REGION Network 19: Panel 19
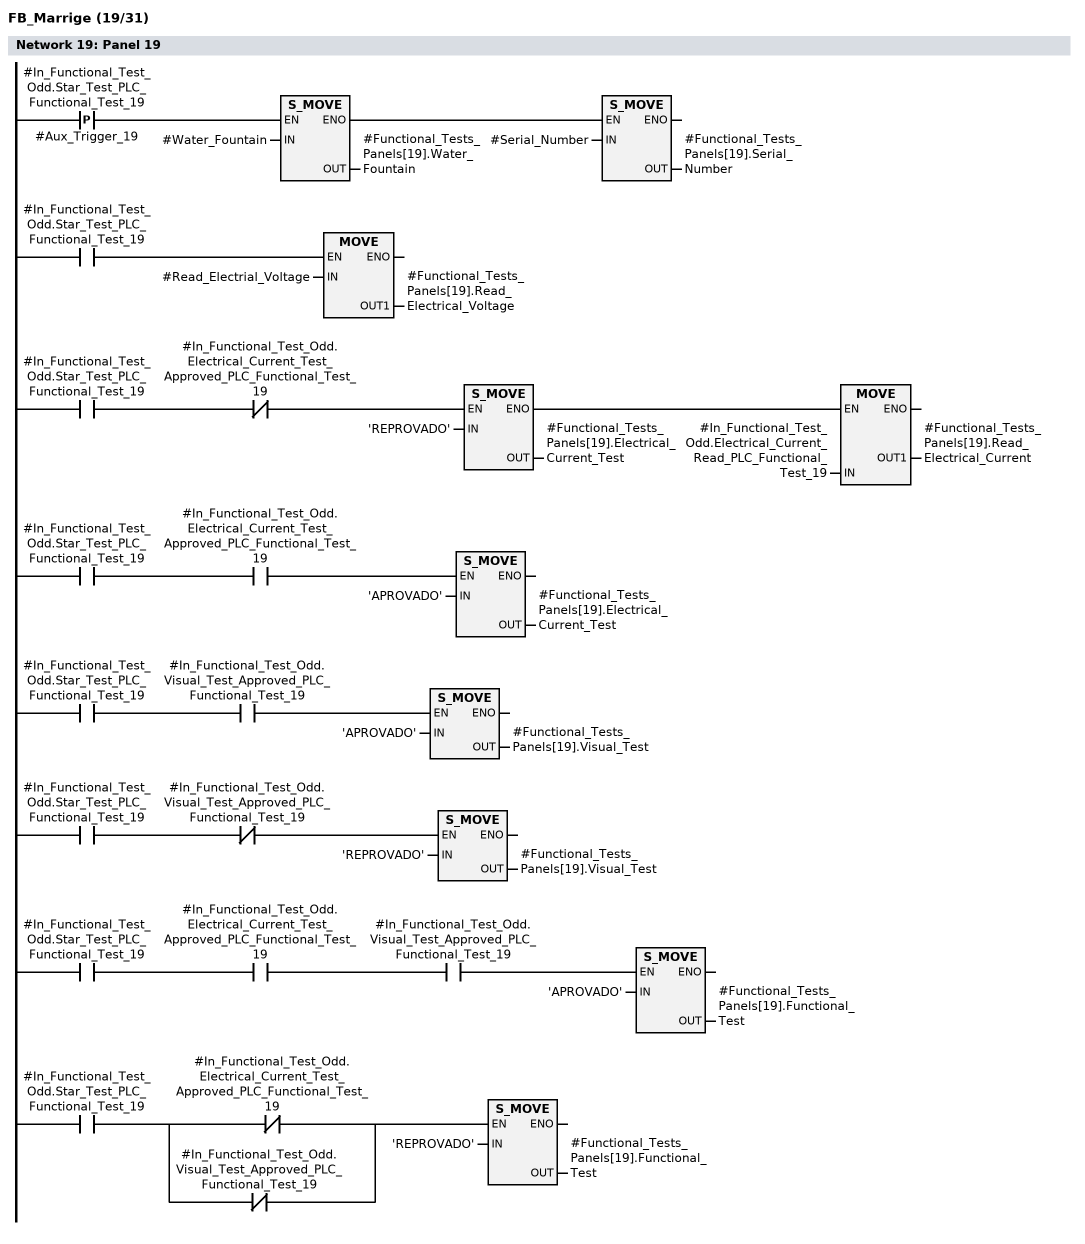
   RUNG wire#powerrail
      P_Contact(operand := #In_Functional_Test_Odd.Star_Test_PLC_Functional_Test_19, bit := #Aux_Trigger_19)
      S_Move(in := #Water_Fountain, out => #Functional_Tests_Panels[19].Water_Fountain)
      S_Move(in := #Serial_Number, out => #Functional_Tests_Panels[19].Serial_Number)
   END_RUNG
   RUNG wire#powerrail
      Contact( #In_Functional_Test_Odd.Star_Test_PLC_Functional_Test_19 )
      Move(in := #Read_Electrial_Voltage, out1 => #Functional_Tests_Panels[19].Read_Electrical_Voltage)
   END_RUNG
   RUNG wire#powerrail
      Contact( #In_Functional_Test_Odd.Star_Test_PLC_Functional_Test_19 )
      I_Contact( #In_Functional_Test_Odd.Electrical_Current_Test_Approved_PLC_Functional_Test_19 )
      S_Move(in := 'REPROVADO', out => #Functional_Tests_Panels[19].Electrical_Current_Test)
      Move(in := #In_Functional_Test_Odd.Electrical_Current_Read_PLC_Functional_Test_19, out1 => #Functional_Tests_Panels[19].Read_Electrical_Current)
   END_RUNG
   RUNG wire#powerrail
      Contact( #In_Functional_Test_Odd.Star_Test_PLC_Functional_Test_19 )
      Contact( #In_Functional_Test_Odd.Electrical_Current_Test_Approved_PLC_Functional_Test_19 )
      S_Move(in := 'APROVADO', out => #Functional_Tests_Panels[19].Electrical_Current_Test)
   END_RUNG
   RUNG wire#powerrail
      Contact( #In_Functional_Test_Odd.Star_Test_PLC_Functional_Test_19 )
      Contact( #In_Functional_Test_Odd.Visual_Test_Approved_PLC_Functional_Test_19 )
      S_Move(in := 'APROVADO', out => #Functional_Tests_Panels[19].Visual_Test)
   END_RUNG
   RUNG wire#powerrail
      Contact( #In_Functional_Test_Odd.Star_Test_PLC_Functional_Test_19 )
      I_Contact( #In_Functional_Test_Odd.Visual_Test_Approved_PLC_Functional_Test_19 )
      S_Move(in := 'REPROVADO', out => #Functional_Tests_Panels[19].Visual_Test)
   END_RUNG
   RUNG wire#powerrail
      Contact( #In_Functional_Test_Odd.Star_Test_PLC_Functional_Test_19 )
      Contact( #In_Functional_Test_Odd.Electrical_Current_Test_Approved_PLC_Functional_Test_19 )
      Contact( #In_Functional_Test_Odd.Visual_Test_Approved_PLC_Functional_Test_19 )
      S_Move(in := 'APROVADO', out => #Functional_Tests_Panels[19].Functional_Test)
   END_RUNG
   RUNG wire#powerrail
      Contact( #In_Functional_Test_Odd.Star_Test_PLC_Functional_Test_19 )
      wire#w1
      I_Contact( #In_Functional_Test_Odd.Electrical_Current_Test_Approved_PLC_Functional_Test_19 )
      wire#w2
      S_Move(in := 'REPROVADO', out => #Functional_Tests_Panels[19].Functional_Test)
   END_RUNG
   RUNG wire#w1
      I_Contact( #In_Functional_Test_Odd.Visual_Test_Approved_PLC_Functional_Test_19 )
   END_RUNG wire#w2
   // the same network as SCL:
   #_w1 := #In_Functional_Test_Odd.Star_Test_PLC_Functional_Test_19 AND NOT #Aux_Trigger_19;   // rising edge of #In_Functional_Test_Odd.Star_Test_PLC_Functional_Test_19
   #Aux_Trigger_19 := #In_Functional_Test_Odd.Star_Test_PLC_Functional_Test_19;
   IF #_w1 THEN
       #Functional_Tests_Panels[19].Water_Fountain := #Water_Fountain;
       #Functional_Tests_Panels[19].Serial_Number := #Serial_Number;
   END_IF;
   IF #In_Functional_Test_Odd.Star_Test_PLC_Functional_Test_19 THEN
       #Functional_Tests_Panels[19].Read_Electrical_Voltage := #Read_Electrial_Voltage;
   END_IF;
   IF #In_Functional_Test_Odd.Star_Test_PLC_Functional_Test_19 AND NOT #In_Functional_Test_Odd.Electrical_Current_Test_Approved_PLC_Functional_Test_19 THEN
       #Functional_Tests_Panels[19].Electrical_Current_Test := 'REPROVADO';
       #Functional_Tests_Panels[19].Read_Electrical_Current := #In_Functional_Test_Odd.Electrical_Current_Read_PLC_Functional_Test_19;
   END_IF;
   IF #In_Functional_Test_Odd.Star_Test_PLC_Functional_Test_19 AND #In_Functional_Test_Odd.Electrical_Current_Test_Approved_PLC_Functional_Test_19 THEN
       #Functional_Tests_Panels[19].Electrical_Current_Test := 'APROVADO';
   END_IF;
   IF #In_Functional_Test_Odd.Star_Test_PLC_Functional_Test_19 AND #In_Functional_Test_Odd.Visual_Test_Approved_PLC_Functional_Test_19 THEN
       #Functional_Tests_Panels[19].Visual_Test := 'APROVADO';
   END_IF;
   IF #In_Functional_Test_Odd.Star_Test_PLC_Functional_Test_19 AND NOT #In_Functional_Test_Odd.Visual_Test_Approved_PLC_Functional_Test_19 THEN
       #Functional_Tests_Panels[19].Visual_Test := 'REPROVADO';
   END_IF;
   IF #In_Functional_Test_Odd.Star_Test_PLC_Functional_Test_19 AND #In_Functional_Test_Odd.Electrical_Current_Test_Approved_PLC_Functional_Test_19 AND #In_Functional_Test_Odd.Visual_Test_Approved_PLC_Functional_Test_19 THEN
       #Functional_Tests_Panels[19].Functional_Test := 'APROVADO';
   END_IF;
   IF #In_Functional_Test_Odd.Star_Test_PLC_Functional_Test_19 AND (NOT #In_Functional_Test_Odd.Electrical_Current_Test_Approved_PLC_Functional_Test_19 OR NOT #In_Functional_Test_Odd.Visual_Test_Approved_PLC_Functional_Test_19) THEN
       #Functional_Tests_Panels[19].Functional_Test := 'REPROVADO';
   END_IF;
END_REGION

REGION Network 20: Panel 20
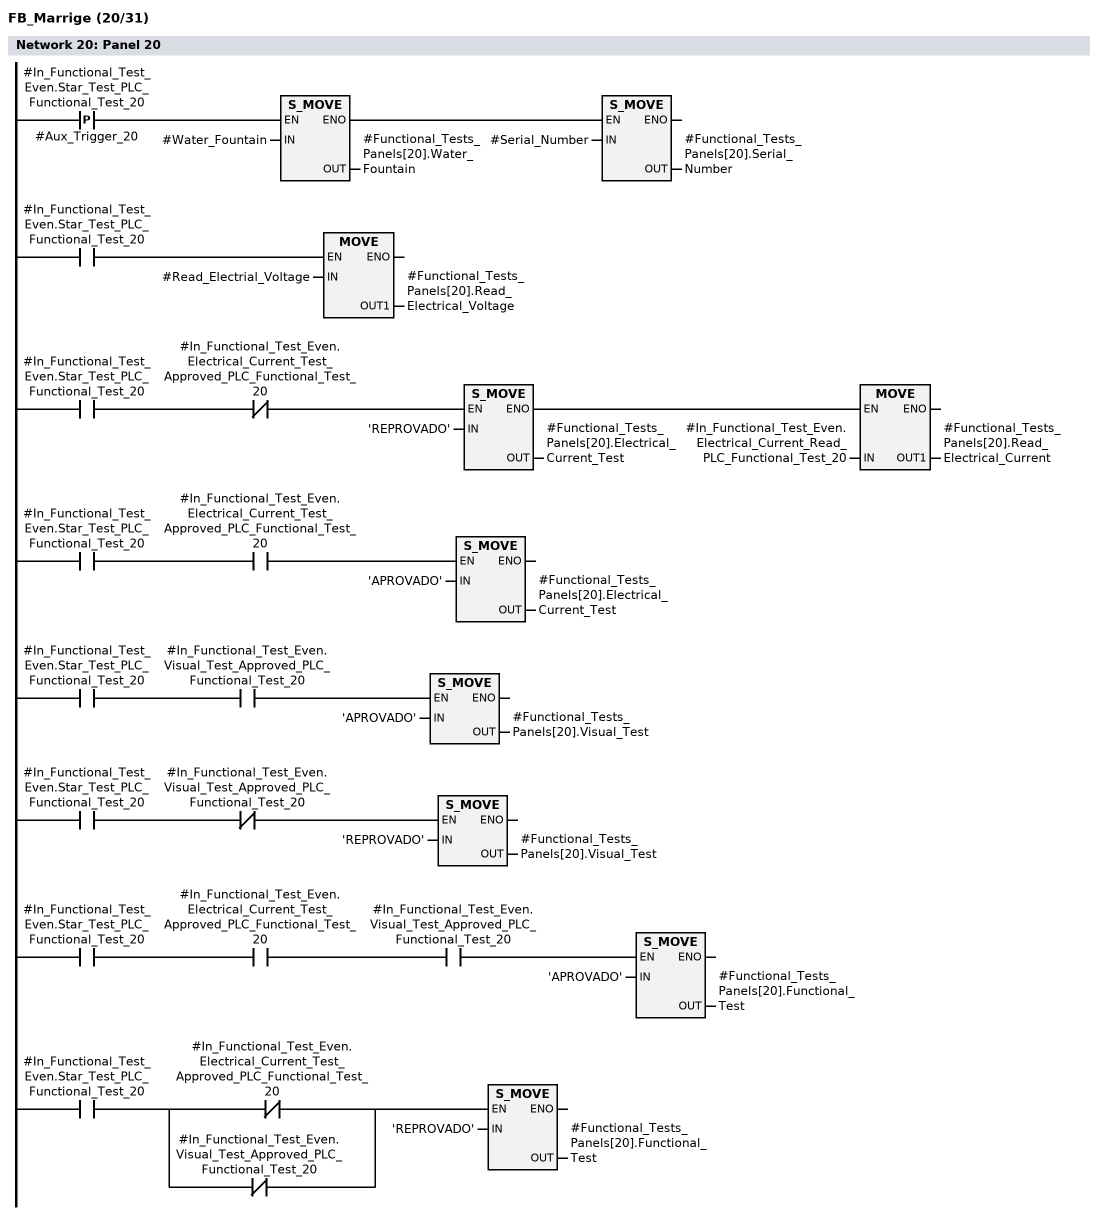
   RUNG wire#powerrail
      P_Contact(operand := #In_Functional_Test_Even.Star_Test_PLC_Functional_Test_20, bit := #Aux_Trigger_20)
      S_Move(in := #Water_Fountain, out => #Functional_Tests_Panels[20].Water_Fountain)
      S_Move(in := #Serial_Number, out => #Functional_Tests_Panels[20].Serial_Number)
   END_RUNG
   RUNG wire#powerrail
      Contact( #In_Functional_Test_Even.Star_Test_PLC_Functional_Test_20 )
      Move(in := #Read_Electrial_Voltage, out1 => #Functional_Tests_Panels[20].Read_Electrical_Voltage)
   END_RUNG
   RUNG wire#powerrail
      Contact( #In_Functional_Test_Even.Star_Test_PLC_Functional_Test_20 )
      I_Contact( #In_Functional_Test_Even.Electrical_Current_Test_Approved_PLC_Functional_Test_20 )
      S_Move(in := 'REPROVADO', out => #Functional_Tests_Panels[20].Electrical_Current_Test)
      Move(in := #In_Functional_Test_Even.Electrical_Current_Read_PLC_Functional_Test_20, out1 => #Functional_Tests_Panels[20].Read_Electrical_Current)
   END_RUNG
   RUNG wire#powerrail
      Contact( #In_Functional_Test_Even.Star_Test_PLC_Functional_Test_20 )
      Contact( #In_Functional_Test_Even.Electrical_Current_Test_Approved_PLC_Functional_Test_20 )
      S_Move(in := 'APROVADO', out => #Functional_Tests_Panels[20].Electrical_Current_Test)
   END_RUNG
   RUNG wire#powerrail
      Contact( #In_Functional_Test_Even.Star_Test_PLC_Functional_Test_20 )
      Contact( #In_Functional_Test_Even.Visual_Test_Approved_PLC_Functional_Test_20 )
      S_Move(in := 'APROVADO', out => #Functional_Tests_Panels[20].Visual_Test)
   END_RUNG
   RUNG wire#powerrail
      Contact( #In_Functional_Test_Even.Star_Test_PLC_Functional_Test_20 )
      I_Contact( #In_Functional_Test_Even.Visual_Test_Approved_PLC_Functional_Test_20 )
      S_Move(in := 'REPROVADO', out => #Functional_Tests_Panels[20].Visual_Test)
   END_RUNG
   RUNG wire#powerrail
      Contact( #In_Functional_Test_Even.Star_Test_PLC_Functional_Test_20 )
      Contact( #In_Functional_Test_Even.Electrical_Current_Test_Approved_PLC_Functional_Test_20 )
      Contact( #In_Functional_Test_Even.Visual_Test_Approved_PLC_Functional_Test_20 )
      S_Move(in := 'APROVADO', out => #Functional_Tests_Panels[20].Functional_Test)
   END_RUNG
   RUNG wire#powerrail
      Contact( #In_Functional_Test_Even.Star_Test_PLC_Functional_Test_20 )
      wire#w1
      I_Contact( #In_Functional_Test_Even.Electrical_Current_Test_Approved_PLC_Functional_Test_20 )
      wire#w2
      S_Move(in := 'REPROVADO', out => #Functional_Tests_Panels[20].Functional_Test)
   END_RUNG
   RUNG wire#w1
      I_Contact( #In_Functional_Test_Even.Visual_Test_Approved_PLC_Functional_Test_20 )
   END_RUNG wire#w2
   // the same network as SCL:
   #_w1 := #In_Functional_Test_Even.Star_Test_PLC_Functional_Test_20 AND NOT #Aux_Trigger_20;   // rising edge of #In_Functional_Test_Even.Star_Test_PLC_Functional_Test_20
   #Aux_Trigger_20 := #In_Functional_Test_Even.Star_Test_PLC_Functional_Test_20;
   IF #_w1 THEN
       #Functional_Tests_Panels[20].Water_Fountain := #Water_Fountain;
       #Functional_Tests_Panels[20].Serial_Number := #Serial_Number;
   END_IF;
   IF #In_Functional_Test_Even.Star_Test_PLC_Functional_Test_20 THEN
       #Functional_Tests_Panels[20].Read_Electrical_Voltage := #Read_Electrial_Voltage;
   END_IF;
   IF #In_Functional_Test_Even.Star_Test_PLC_Functional_Test_20 AND NOT #In_Functional_Test_Even.Electrical_Current_Test_Approved_PLC_Functional_Test_20 THEN
       #Functional_Tests_Panels[20].Electrical_Current_Test := 'REPROVADO';
       #Functional_Tests_Panels[20].Read_Electrical_Current := #In_Functional_Test_Even.Electrical_Current_Read_PLC_Functional_Test_20;
   END_IF;
   IF #In_Functional_Test_Even.Star_Test_PLC_Functional_Test_20 AND #In_Functional_Test_Even.Electrical_Current_Test_Approved_PLC_Functional_Test_20 THEN
       #Functional_Tests_Panels[20].Electrical_Current_Test := 'APROVADO';
   END_IF;
   IF #In_Functional_Test_Even.Star_Test_PLC_Functional_Test_20 AND #In_Functional_Test_Even.Visual_Test_Approved_PLC_Functional_Test_20 THEN
       #Functional_Tests_Panels[20].Visual_Test := 'APROVADO';
   END_IF;
   IF #In_Functional_Test_Even.Star_Test_PLC_Functional_Test_20 AND NOT #In_Functional_Test_Even.Visual_Test_Approved_PLC_Functional_Test_20 THEN
       #Functional_Tests_Panels[20].Visual_Test := 'REPROVADO';
   END_IF;
   IF #In_Functional_Test_Even.Star_Test_PLC_Functional_Test_20 AND #In_Functional_Test_Even.Electrical_Current_Test_Approved_PLC_Functional_Test_20 AND #In_Functional_Test_Even.Visual_Test_Approved_PLC_Functional_Test_20 THEN
       #Functional_Tests_Panels[20].Functional_Test := 'APROVADO';
   END_IF;
   IF #In_Functional_Test_Even.Star_Test_PLC_Functional_Test_20 AND (NOT #In_Functional_Test_Even.Electrical_Current_Test_Approved_PLC_Functional_Test_20 OR NOT #In_Functional_Test_Even.Visual_Test_Approved_PLC_Functional_Test_20) THEN
       #Functional_Tests_Panels[20].Functional_Test := 'REPROVADO';
   END_IF;
END_REGION

REGION Network 21: Panel 21
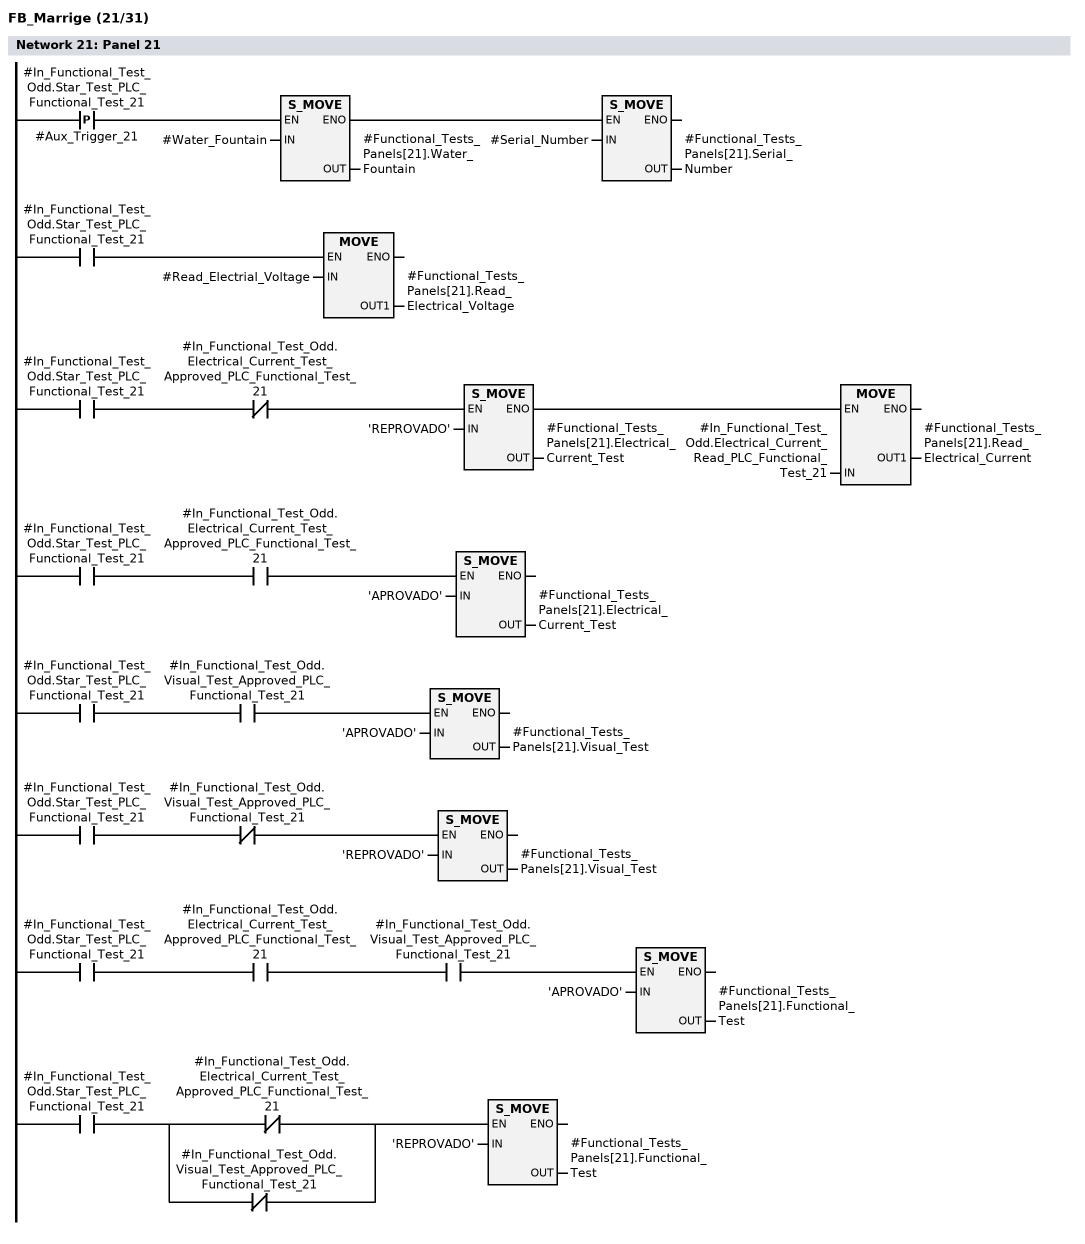
   RUNG wire#powerrail
      P_Contact(operand := #In_Functional_Test_Odd.Star_Test_PLC_Functional_Test_21, bit := #Aux_Trigger_21)
      S_Move(in := #Water_Fountain, out => #Functional_Tests_Panels[21].Water_Fountain)
      S_Move(in := #Serial_Number, out => #Functional_Tests_Panels[21].Serial_Number)
   END_RUNG
   RUNG wire#powerrail
      Contact( #In_Functional_Test_Odd.Star_Test_PLC_Functional_Test_21 )
      Move(in := #Read_Electrial_Voltage, out1 => #Functional_Tests_Panels[21].Read_Electrical_Voltage)
   END_RUNG
   RUNG wire#powerrail
      Contact( #In_Functional_Test_Odd.Star_Test_PLC_Functional_Test_21 )
      I_Contact( #In_Functional_Test_Odd.Electrical_Current_Test_Approved_PLC_Functional_Test_21 )
      S_Move(in := 'REPROVADO', out => #Functional_Tests_Panels[21].Electrical_Current_Test)
      Move(in := #In_Functional_Test_Odd.Electrical_Current_Read_PLC_Functional_Test_21, out1 => #Functional_Tests_Panels[21].Read_Electrical_Current)
   END_RUNG
   RUNG wire#powerrail
      Contact( #In_Functional_Test_Odd.Star_Test_PLC_Functional_Test_21 )
      Contact( #In_Functional_Test_Odd.Electrical_Current_Test_Approved_PLC_Functional_Test_21 )
      S_Move(in := 'APROVADO', out => #Functional_Tests_Panels[21].Electrical_Current_Test)
   END_RUNG
   RUNG wire#powerrail
      Contact( #In_Functional_Test_Odd.Star_Test_PLC_Functional_Test_21 )
      Contact( #In_Functional_Test_Odd.Visual_Test_Approved_PLC_Functional_Test_21 )
      S_Move(in := 'APROVADO', out => #Functional_Tests_Panels[21].Visual_Test)
   END_RUNG
   RUNG wire#powerrail
      Contact( #In_Functional_Test_Odd.Star_Test_PLC_Functional_Test_21 )
      I_Contact( #In_Functional_Test_Odd.Visual_Test_Approved_PLC_Functional_Test_21 )
      S_Move(in := 'REPROVADO', out => #Functional_Tests_Panels[21].Visual_Test)
   END_RUNG
   RUNG wire#powerrail
      Contact( #In_Functional_Test_Odd.Star_Test_PLC_Functional_Test_21 )
      Contact( #In_Functional_Test_Odd.Electrical_Current_Test_Approved_PLC_Functional_Test_21 )
      Contact( #In_Functional_Test_Odd.Visual_Test_Approved_PLC_Functional_Test_21 )
      S_Move(in := 'APROVADO', out => #Functional_Tests_Panels[21].Functional_Test)
   END_RUNG
   RUNG wire#powerrail
      Contact( #In_Functional_Test_Odd.Star_Test_PLC_Functional_Test_21 )
      wire#w1
      I_Contact( #In_Functional_Test_Odd.Electrical_Current_Test_Approved_PLC_Functional_Test_21 )
      wire#w2
      S_Move(in := 'REPROVADO', out => #Functional_Tests_Panels[21].Functional_Test)
   END_RUNG
   RUNG wire#w1
      I_Contact( #In_Functional_Test_Odd.Visual_Test_Approved_PLC_Functional_Test_21 )
   END_RUNG wire#w2
   // the same network as SCL:
   #_w1 := #In_Functional_Test_Odd.Star_Test_PLC_Functional_Test_21 AND NOT #Aux_Trigger_21;   // rising edge of #In_Functional_Test_Odd.Star_Test_PLC_Functional_Test_21
   #Aux_Trigger_21 := #In_Functional_Test_Odd.Star_Test_PLC_Functional_Test_21;
   IF #_w1 THEN
       #Functional_Tests_Panels[21].Water_Fountain := #Water_Fountain;
       #Functional_Tests_Panels[21].Serial_Number := #Serial_Number;
   END_IF;
   IF #In_Functional_Test_Odd.Star_Test_PLC_Functional_Test_21 THEN
       #Functional_Tests_Panels[21].Read_Electrical_Voltage := #Read_Electrial_Voltage;
   END_IF;
   IF #In_Functional_Test_Odd.Star_Test_PLC_Functional_Test_21 AND NOT #In_Functional_Test_Odd.Electrical_Current_Test_Approved_PLC_Functional_Test_21 THEN
       #Functional_Tests_Panels[21].Electrical_Current_Test := 'REPROVADO';
       #Functional_Tests_Panels[21].Read_Electrical_Current := #In_Functional_Test_Odd.Electrical_Current_Read_PLC_Functional_Test_21;
   END_IF;
   IF #In_Functional_Test_Odd.Star_Test_PLC_Functional_Test_21 AND #In_Functional_Test_Odd.Electrical_Current_Test_Approved_PLC_Functional_Test_21 THEN
       #Functional_Tests_Panels[21].Electrical_Current_Test := 'APROVADO';
   END_IF;
   IF #In_Functional_Test_Odd.Star_Test_PLC_Functional_Test_21 AND #In_Functional_Test_Odd.Visual_Test_Approved_PLC_Functional_Test_21 THEN
       #Functional_Tests_Panels[21].Visual_Test := 'APROVADO';
   END_IF;
   IF #In_Functional_Test_Odd.Star_Test_PLC_Functional_Test_21 AND NOT #In_Functional_Test_Odd.Visual_Test_Approved_PLC_Functional_Test_21 THEN
       #Functional_Tests_Panels[21].Visual_Test := 'REPROVADO';
   END_IF;
   IF #In_Functional_Test_Odd.Star_Test_PLC_Functional_Test_21 AND #In_Functional_Test_Odd.Electrical_Current_Test_Approved_PLC_Functional_Test_21 AND #In_Functional_Test_Odd.Visual_Test_Approved_PLC_Functional_Test_21 THEN
       #Functional_Tests_Panels[21].Functional_Test := 'APROVADO';
   END_IF;
   IF #In_Functional_Test_Odd.Star_Test_PLC_Functional_Test_21 AND (NOT #In_Functional_Test_Odd.Electrical_Current_Test_Approved_PLC_Functional_Test_21 OR NOT #In_Functional_Test_Odd.Visual_Test_Approved_PLC_Functional_Test_21) THEN
       #Functional_Tests_Panels[21].Functional_Test := 'REPROVADO';
   END_IF;
END_REGION

REGION Network 22: Panel 22
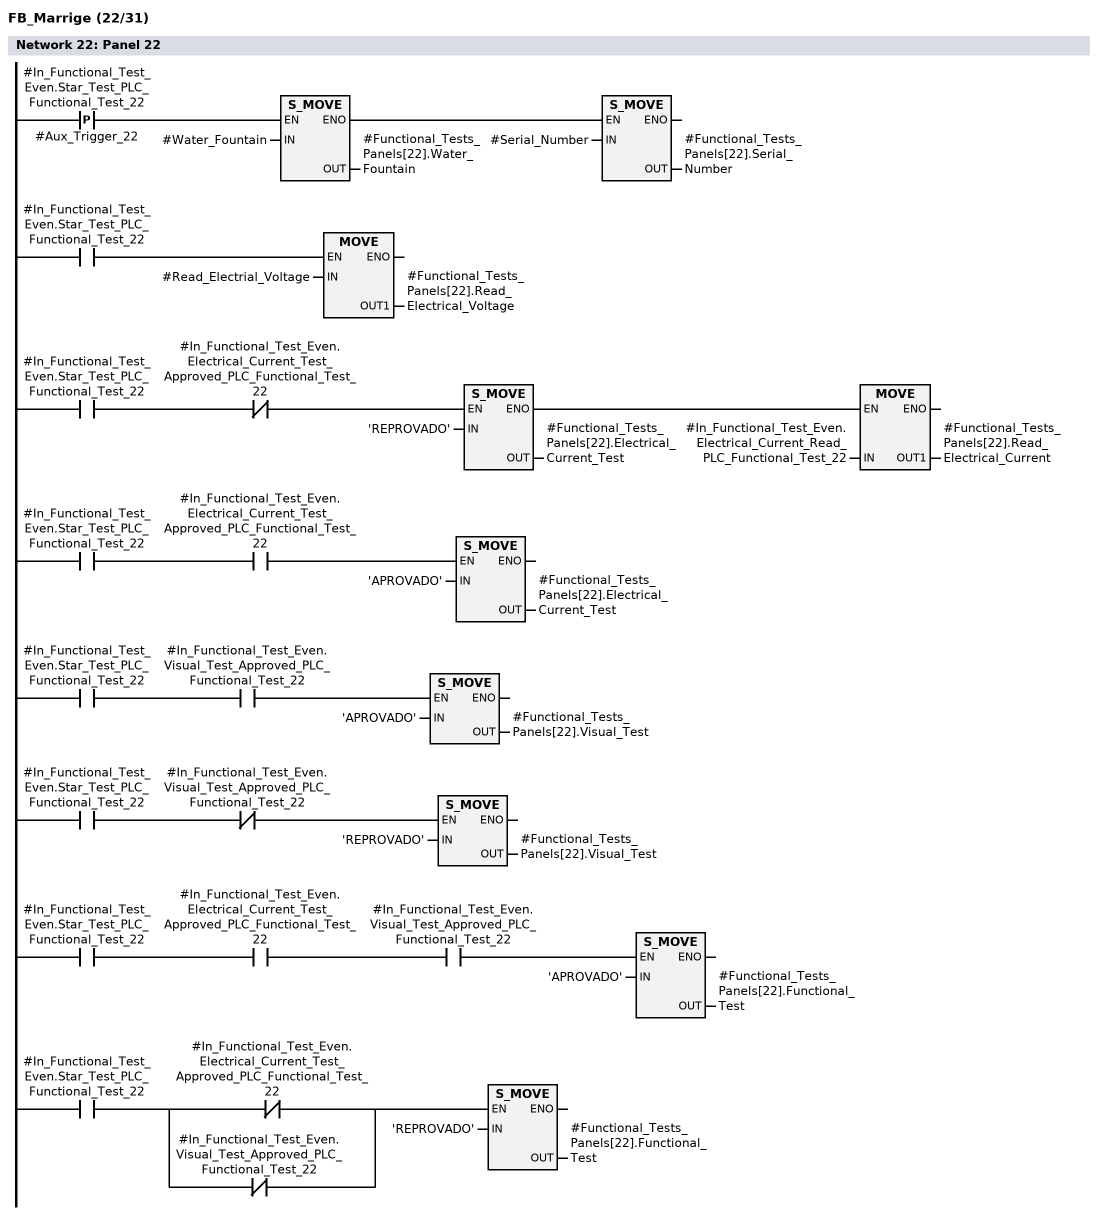
   RUNG wire#powerrail
      P_Contact(operand := #In_Functional_Test_Even.Star_Test_PLC_Functional_Test_22, bit := #Aux_Trigger_22)
      S_Move(in := #Water_Fountain, out => #Functional_Tests_Panels[22].Water_Fountain)
      S_Move(in := #Serial_Number, out => #Functional_Tests_Panels[22].Serial_Number)
   END_RUNG
   RUNG wire#powerrail
      Contact( #In_Functional_Test_Even.Star_Test_PLC_Functional_Test_22 )
      Move(in := #Read_Electrial_Voltage, out1 => #Functional_Tests_Panels[22].Read_Electrical_Voltage)
   END_RUNG
   RUNG wire#powerrail
      Contact( #In_Functional_Test_Even.Star_Test_PLC_Functional_Test_22 )
      I_Contact( #In_Functional_Test_Even.Electrical_Current_Test_Approved_PLC_Functional_Test_22 )
      S_Move(in := 'REPROVADO', out => #Functional_Tests_Panels[22].Electrical_Current_Test)
      Move(in := #In_Functional_Test_Even.Electrical_Current_Read_PLC_Functional_Test_22, out1 => #Functional_Tests_Panels[22].Read_Electrical_Current)
   END_RUNG
   RUNG wire#powerrail
      Contact( #In_Functional_Test_Even.Star_Test_PLC_Functional_Test_22 )
      Contact( #In_Functional_Test_Even.Electrical_Current_Test_Approved_PLC_Functional_Test_22 )
      S_Move(in := 'APROVADO', out => #Functional_Tests_Panels[22].Electrical_Current_Test)
   END_RUNG
   RUNG wire#powerrail
      Contact( #In_Functional_Test_Even.Star_Test_PLC_Functional_Test_22 )
      Contact( #In_Functional_Test_Even.Visual_Test_Approved_PLC_Functional_Test_22 )
      S_Move(in := 'APROVADO', out => #Functional_Tests_Panels[22].Visual_Test)
   END_RUNG
   RUNG wire#powerrail
      Contact( #In_Functional_Test_Even.Star_Test_PLC_Functional_Test_22 )
      I_Contact( #In_Functional_Test_Even.Visual_Test_Approved_PLC_Functional_Test_22 )
      S_Move(in := 'REPROVADO', out => #Functional_Tests_Panels[22].Visual_Test)
   END_RUNG
   RUNG wire#powerrail
      Contact( #In_Functional_Test_Even.Star_Test_PLC_Functional_Test_22 )
      Contact( #In_Functional_Test_Even.Electrical_Current_Test_Approved_PLC_Functional_Test_22 )
      Contact( #In_Functional_Test_Even.Visual_Test_Approved_PLC_Functional_Test_22 )
      S_Move(in := 'APROVADO', out => #Functional_Tests_Panels[22].Functional_Test)
   END_RUNG
   RUNG wire#powerrail
      Contact( #In_Functional_Test_Even.Star_Test_PLC_Functional_Test_22 )
      wire#w1
      I_Contact( #In_Functional_Test_Even.Electrical_Current_Test_Approved_PLC_Functional_Test_22 )
      wire#w2
      S_Move(in := 'REPROVADO', out => #Functional_Tests_Panels[22].Functional_Test)
   END_RUNG
   RUNG wire#w1
      I_Contact( #In_Functional_Test_Even.Visual_Test_Approved_PLC_Functional_Test_22 )
   END_RUNG wire#w2
   // the same network as SCL:
   #_w1 := #In_Functional_Test_Even.Star_Test_PLC_Functional_Test_22 AND NOT #Aux_Trigger_22;   // rising edge of #In_Functional_Test_Even.Star_Test_PLC_Functional_Test_22
   #Aux_Trigger_22 := #In_Functional_Test_Even.Star_Test_PLC_Functional_Test_22;
   IF #_w1 THEN
       #Functional_Tests_Panels[22].Water_Fountain := #Water_Fountain;
       #Functional_Tests_Panels[22].Serial_Number := #Serial_Number;
   END_IF;
   IF #In_Functional_Test_Even.Star_Test_PLC_Functional_Test_22 THEN
       #Functional_Tests_Panels[22].Read_Electrical_Voltage := #Read_Electrial_Voltage;
   END_IF;
   IF #In_Functional_Test_Even.Star_Test_PLC_Functional_Test_22 AND NOT #In_Functional_Test_Even.Electrical_Current_Test_Approved_PLC_Functional_Test_22 THEN
       #Functional_Tests_Panels[22].Electrical_Current_Test := 'REPROVADO';
       #Functional_Tests_Panels[22].Read_Electrical_Current := #In_Functional_Test_Even.Electrical_Current_Read_PLC_Functional_Test_22;
   END_IF;
   IF #In_Functional_Test_Even.Star_Test_PLC_Functional_Test_22 AND #In_Functional_Test_Even.Electrical_Current_Test_Approved_PLC_Functional_Test_22 THEN
       #Functional_Tests_Panels[22].Electrical_Current_Test := 'APROVADO';
   END_IF;
   IF #In_Functional_Test_Even.Star_Test_PLC_Functional_Test_22 AND #In_Functional_Test_Even.Visual_Test_Approved_PLC_Functional_Test_22 THEN
       #Functional_Tests_Panels[22].Visual_Test := 'APROVADO';
   END_IF;
   IF #In_Functional_Test_Even.Star_Test_PLC_Functional_Test_22 AND NOT #In_Functional_Test_Even.Visual_Test_Approved_PLC_Functional_Test_22 THEN
       #Functional_Tests_Panels[22].Visual_Test := 'REPROVADO';
   END_IF;
   IF #In_Functional_Test_Even.Star_Test_PLC_Functional_Test_22 AND #In_Functional_Test_Even.Electrical_Current_Test_Approved_PLC_Functional_Test_22 AND #In_Functional_Test_Even.Visual_Test_Approved_PLC_Functional_Test_22 THEN
       #Functional_Tests_Panels[22].Functional_Test := 'APROVADO';
   END_IF;
   IF #In_Functional_Test_Even.Star_Test_PLC_Functional_Test_22 AND (NOT #In_Functional_Test_Even.Electrical_Current_Test_Approved_PLC_Functional_Test_22 OR NOT #In_Functional_Test_Even.Visual_Test_Approved_PLC_Functional_Test_22) THEN
       #Functional_Tests_Panels[22].Functional_Test := 'REPROVADO';
   END_IF;
END_REGION

REGION Network 23: Panel 23
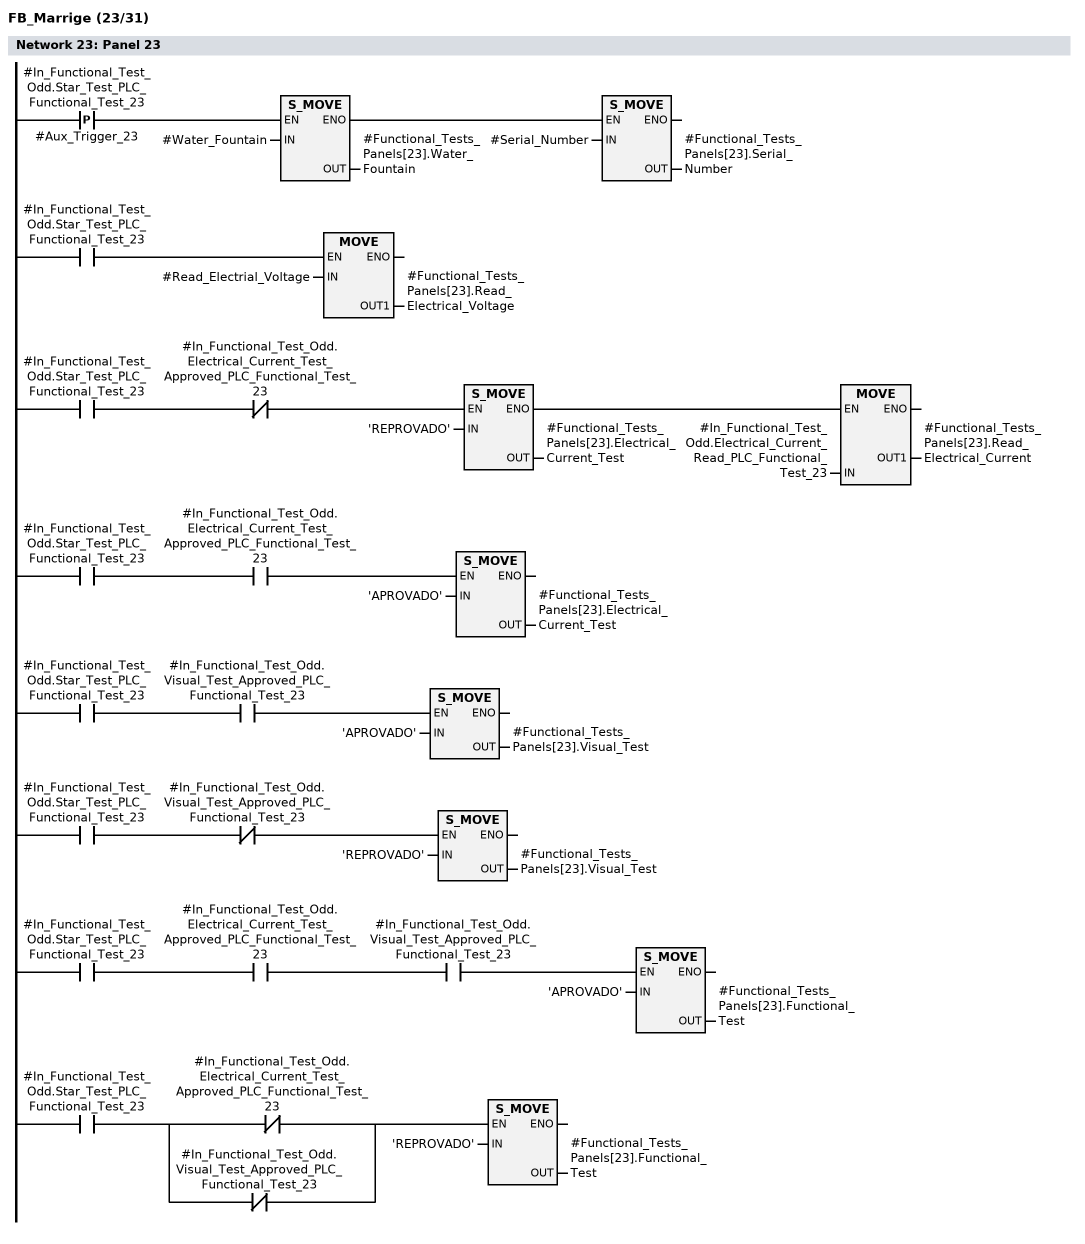
   RUNG wire#powerrail
      P_Contact(operand := #In_Functional_Test_Odd.Star_Test_PLC_Functional_Test_23, bit := #Aux_Trigger_23)
      S_Move(in := #Water_Fountain, out => #Functional_Tests_Panels[23].Water_Fountain)
      S_Move(in := #Serial_Number, out => #Functional_Tests_Panels[23].Serial_Number)
   END_RUNG
   RUNG wire#powerrail
      Contact( #In_Functional_Test_Odd.Star_Test_PLC_Functional_Test_23 )
      Move(in := #Read_Electrial_Voltage, out1 => #Functional_Tests_Panels[23].Read_Electrical_Voltage)
   END_RUNG
   RUNG wire#powerrail
      Contact( #In_Functional_Test_Odd.Star_Test_PLC_Functional_Test_23 )
      I_Contact( #In_Functional_Test_Odd.Electrical_Current_Test_Approved_PLC_Functional_Test_23 )
      S_Move(in := 'REPROVADO', out => #Functional_Tests_Panels[23].Electrical_Current_Test)
      Move(in := #In_Functional_Test_Odd.Electrical_Current_Read_PLC_Functional_Test_23, out1 => #Functional_Tests_Panels[23].Read_Electrical_Current)
   END_RUNG
   RUNG wire#powerrail
      Contact( #In_Functional_Test_Odd.Star_Test_PLC_Functional_Test_23 )
      Contact( #In_Functional_Test_Odd.Electrical_Current_Test_Approved_PLC_Functional_Test_23 )
      S_Move(in := 'APROVADO', out => #Functional_Tests_Panels[23].Electrical_Current_Test)
   END_RUNG
   RUNG wire#powerrail
      Contact( #In_Functional_Test_Odd.Star_Test_PLC_Functional_Test_23 )
      Contact( #In_Functional_Test_Odd.Visual_Test_Approved_PLC_Functional_Test_23 )
      S_Move(in := 'APROVADO', out => #Functional_Tests_Panels[23].Visual_Test)
   END_RUNG
   RUNG wire#powerrail
      Contact( #In_Functional_Test_Odd.Star_Test_PLC_Functional_Test_23 )
      I_Contact( #In_Functional_Test_Odd.Visual_Test_Approved_PLC_Functional_Test_23 )
      S_Move(in := 'REPROVADO', out => #Functional_Tests_Panels[23].Visual_Test)
   END_RUNG
   RUNG wire#powerrail
      Contact( #In_Functional_Test_Odd.Star_Test_PLC_Functional_Test_23 )
      Contact( #In_Functional_Test_Odd.Electrical_Current_Test_Approved_PLC_Functional_Test_23 )
      Contact( #In_Functional_Test_Odd.Visual_Test_Approved_PLC_Functional_Test_23 )
      S_Move(in := 'APROVADO', out => #Functional_Tests_Panels[23].Functional_Test)
   END_RUNG
   RUNG wire#powerrail
      Contact( #In_Functional_Test_Odd.Star_Test_PLC_Functional_Test_23 )
      wire#w1
      I_Contact( #In_Functional_Test_Odd.Electrical_Current_Test_Approved_PLC_Functional_Test_23 )
      wire#w2
      S_Move(in := 'REPROVADO', out => #Functional_Tests_Panels[23].Functional_Test)
   END_RUNG
   RUNG wire#w1
      I_Contact( #In_Functional_Test_Odd.Visual_Test_Approved_PLC_Functional_Test_23 )
   END_RUNG wire#w2
   // the same network as SCL:
   #_w1 := #In_Functional_Test_Odd.Star_Test_PLC_Functional_Test_23 AND NOT #Aux_Trigger_23;   // rising edge of #In_Functional_Test_Odd.Star_Test_PLC_Functional_Test_23
   #Aux_Trigger_23 := #In_Functional_Test_Odd.Star_Test_PLC_Functional_Test_23;
   IF #_w1 THEN
       #Functional_Tests_Panels[23].Water_Fountain := #Water_Fountain;
       #Functional_Tests_Panels[23].Serial_Number := #Serial_Number;
   END_IF;
   IF #In_Functional_Test_Odd.Star_Test_PLC_Functional_Test_23 THEN
       #Functional_Tests_Panels[23].Read_Electrical_Voltage := #Read_Electrial_Voltage;
   END_IF;
   IF #In_Functional_Test_Odd.Star_Test_PLC_Functional_Test_23 AND NOT #In_Functional_Test_Odd.Electrical_Current_Test_Approved_PLC_Functional_Test_23 THEN
       #Functional_Tests_Panels[23].Electrical_Current_Test := 'REPROVADO';
       #Functional_Tests_Panels[23].Read_Electrical_Current := #In_Functional_Test_Odd.Electrical_Current_Read_PLC_Functional_Test_23;
   END_IF;
   IF #In_Functional_Test_Odd.Star_Test_PLC_Functional_Test_23 AND #In_Functional_Test_Odd.Electrical_Current_Test_Approved_PLC_Functional_Test_23 THEN
       #Functional_Tests_Panels[23].Electrical_Current_Test := 'APROVADO';
   END_IF;
   IF #In_Functional_Test_Odd.Star_Test_PLC_Functional_Test_23 AND #In_Functional_Test_Odd.Visual_Test_Approved_PLC_Functional_Test_23 THEN
       #Functional_Tests_Panels[23].Visual_Test := 'APROVADO';
   END_IF;
   IF #In_Functional_Test_Odd.Star_Test_PLC_Functional_Test_23 AND NOT #In_Functional_Test_Odd.Visual_Test_Approved_PLC_Functional_Test_23 THEN
       #Functional_Tests_Panels[23].Visual_Test := 'REPROVADO';
   END_IF;
   IF #In_Functional_Test_Odd.Star_Test_PLC_Functional_Test_23 AND #In_Functional_Test_Odd.Electrical_Current_Test_Approved_PLC_Functional_Test_23 AND #In_Functional_Test_Odd.Visual_Test_Approved_PLC_Functional_Test_23 THEN
       #Functional_Tests_Panels[23].Functional_Test := 'APROVADO';
   END_IF;
   IF #In_Functional_Test_Odd.Star_Test_PLC_Functional_Test_23 AND (NOT #In_Functional_Test_Odd.Electrical_Current_Test_Approved_PLC_Functional_Test_23 OR NOT #In_Functional_Test_Odd.Visual_Test_Approved_PLC_Functional_Test_23) THEN
       #Functional_Tests_Panels[23].Functional_Test := 'REPROVADO';
   END_IF;
END_REGION

REGION Network 24: Panel 24
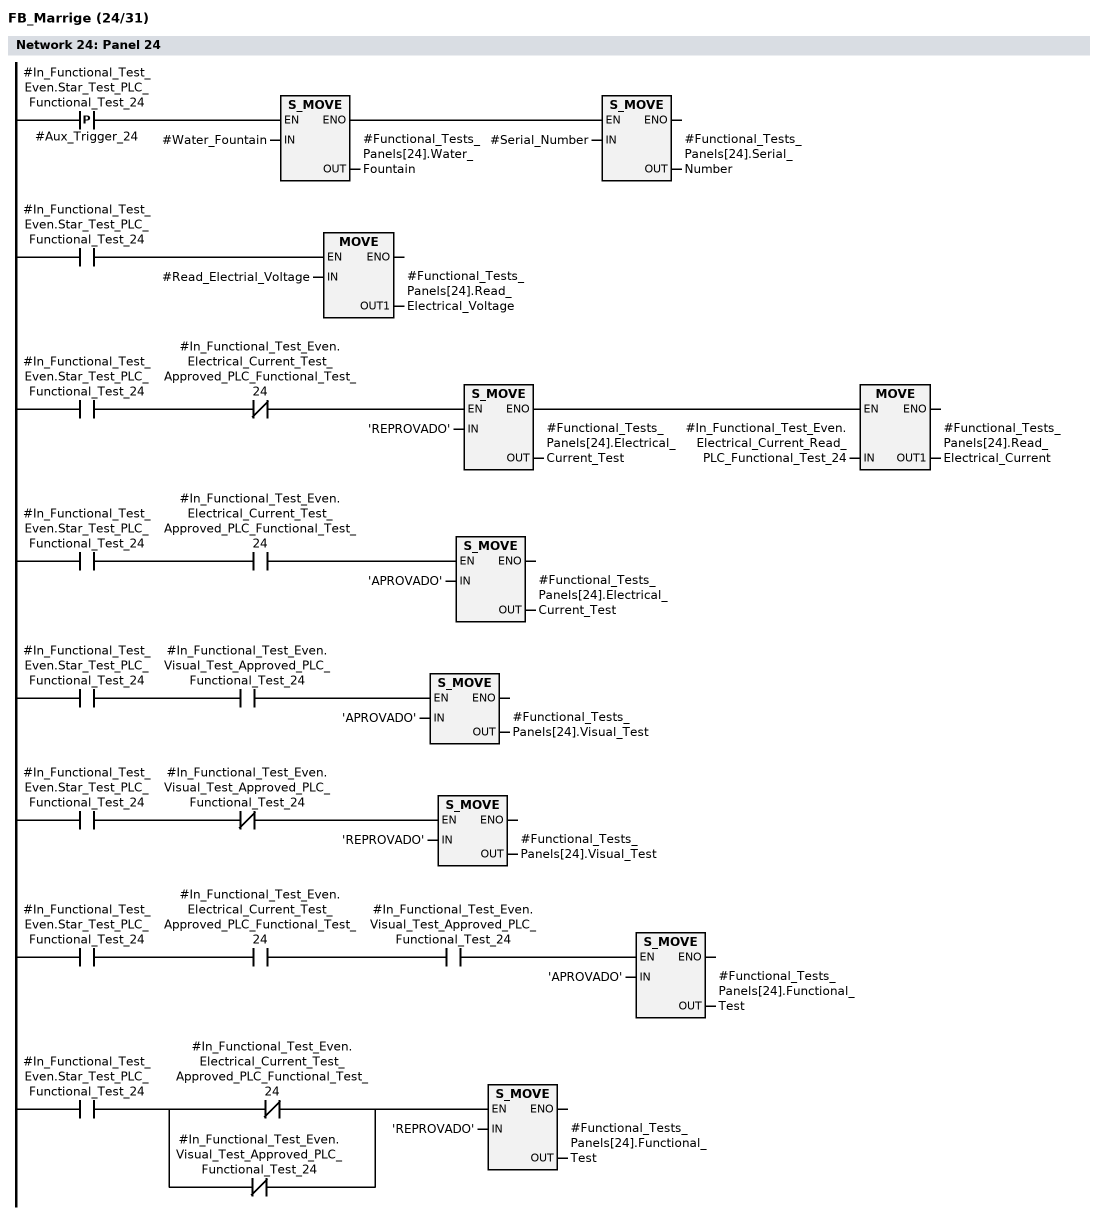
   RUNG wire#powerrail
      P_Contact(operand := #In_Functional_Test_Even.Star_Test_PLC_Functional_Test_24, bit := #Aux_Trigger_24)
      S_Move(in := #Water_Fountain, out => #Functional_Tests_Panels[24].Water_Fountain)
      S_Move(in := #Serial_Number, out => #Functional_Tests_Panels[24].Serial_Number)
   END_RUNG
   RUNG wire#powerrail
      Contact( #In_Functional_Test_Even.Star_Test_PLC_Functional_Test_24 )
      Move(in := #Read_Electrial_Voltage, out1 => #Functional_Tests_Panels[24].Read_Electrical_Voltage)
   END_RUNG
   RUNG wire#powerrail
      Contact( #In_Functional_Test_Even.Star_Test_PLC_Functional_Test_24 )
      I_Contact( #In_Functional_Test_Even.Electrical_Current_Test_Approved_PLC_Functional_Test_24 )
      S_Move(in := 'REPROVADO', out => #Functional_Tests_Panels[24].Electrical_Current_Test)
      Move(in := #In_Functional_Test_Even.Electrical_Current_Read_PLC_Functional_Test_24, out1 => #Functional_Tests_Panels[24].Read_Electrical_Current)
   END_RUNG
   RUNG wire#powerrail
      Contact( #In_Functional_Test_Even.Star_Test_PLC_Functional_Test_24 )
      Contact( #In_Functional_Test_Even.Electrical_Current_Test_Approved_PLC_Functional_Test_24 )
      S_Move(in := 'APROVADO', out => #Functional_Tests_Panels[24].Electrical_Current_Test)
   END_RUNG
   RUNG wire#powerrail
      Contact( #In_Functional_Test_Even.Star_Test_PLC_Functional_Test_24 )
      Contact( #In_Functional_Test_Even.Visual_Test_Approved_PLC_Functional_Test_24 )
      S_Move(in := 'APROVADO', out => #Functional_Tests_Panels[24].Visual_Test)
   END_RUNG
   RUNG wire#powerrail
      Contact( #In_Functional_Test_Even.Star_Test_PLC_Functional_Test_24 )
      I_Contact( #In_Functional_Test_Even.Visual_Test_Approved_PLC_Functional_Test_24 )
      S_Move(in := 'REPROVADO', out => #Functional_Tests_Panels[24].Visual_Test)
   END_RUNG
   RUNG wire#powerrail
      Contact( #In_Functional_Test_Even.Star_Test_PLC_Functional_Test_24 )
      Contact( #In_Functional_Test_Even.Electrical_Current_Test_Approved_PLC_Functional_Test_24 )
      Contact( #In_Functional_Test_Even.Visual_Test_Approved_PLC_Functional_Test_24 )
      S_Move(in := 'APROVADO', out => #Functional_Tests_Panels[24].Functional_Test)
   END_RUNG
   RUNG wire#powerrail
      Contact( #In_Functional_Test_Even.Star_Test_PLC_Functional_Test_24 )
      wire#w1
      I_Contact( #In_Functional_Test_Even.Electrical_Current_Test_Approved_PLC_Functional_Test_24 )
      wire#w2
      S_Move(in := 'REPROVADO', out => #Functional_Tests_Panels[24].Functional_Test)
   END_RUNG
   RUNG wire#w1
      I_Contact( #In_Functional_Test_Even.Visual_Test_Approved_PLC_Functional_Test_24 )
   END_RUNG wire#w2
   // the same network as SCL:
   #_w1 := #In_Functional_Test_Even.Star_Test_PLC_Functional_Test_24 AND NOT #Aux_Trigger_24;   // rising edge of #In_Functional_Test_Even.Star_Test_PLC_Functional_Test_24
   #Aux_Trigger_24 := #In_Functional_Test_Even.Star_Test_PLC_Functional_Test_24;
   IF #_w1 THEN
       #Functional_Tests_Panels[24].Water_Fountain := #Water_Fountain;
       #Functional_Tests_Panels[24].Serial_Number := #Serial_Number;
   END_IF;
   IF #In_Functional_Test_Even.Star_Test_PLC_Functional_Test_24 THEN
       #Functional_Tests_Panels[24].Read_Electrical_Voltage := #Read_Electrial_Voltage;
   END_IF;
   IF #In_Functional_Test_Even.Star_Test_PLC_Functional_Test_24 AND NOT #In_Functional_Test_Even.Electrical_Current_Test_Approved_PLC_Functional_Test_24 THEN
       #Functional_Tests_Panels[24].Electrical_Current_Test := 'REPROVADO';
       #Functional_Tests_Panels[24].Read_Electrical_Current := #In_Functional_Test_Even.Electrical_Current_Read_PLC_Functional_Test_24;
   END_IF;
   IF #In_Functional_Test_Even.Star_Test_PLC_Functional_Test_24 AND #In_Functional_Test_Even.Electrical_Current_Test_Approved_PLC_Functional_Test_24 THEN
       #Functional_Tests_Panels[24].Electrical_Current_Test := 'APROVADO';
   END_IF;
   IF #In_Functional_Test_Even.Star_Test_PLC_Functional_Test_24 AND #In_Functional_Test_Even.Visual_Test_Approved_PLC_Functional_Test_24 THEN
       #Functional_Tests_Panels[24].Visual_Test := 'APROVADO';
   END_IF;
   IF #In_Functional_Test_Even.Star_Test_PLC_Functional_Test_24 AND NOT #In_Functional_Test_Even.Visual_Test_Approved_PLC_Functional_Test_24 THEN
       #Functional_Tests_Panels[24].Visual_Test := 'REPROVADO';
   END_IF;
   IF #In_Functional_Test_Even.Star_Test_PLC_Functional_Test_24 AND #In_Functional_Test_Even.Electrical_Current_Test_Approved_PLC_Functional_Test_24 AND #In_Functional_Test_Even.Visual_Test_Approved_PLC_Functional_Test_24 THEN
       #Functional_Tests_Panels[24].Functional_Test := 'APROVADO';
   END_IF;
   IF #In_Functional_Test_Even.Star_Test_PLC_Functional_Test_24 AND (NOT #In_Functional_Test_Even.Electrical_Current_Test_Approved_PLC_Functional_Test_24 OR NOT #In_Functional_Test_Even.Visual_Test_Approved_PLC_Functional_Test_24) THEN
       #Functional_Tests_Panels[24].Functional_Test := 'REPROVADO';
   END_IF;
END_REGION

REGION Network 25: Panel 25
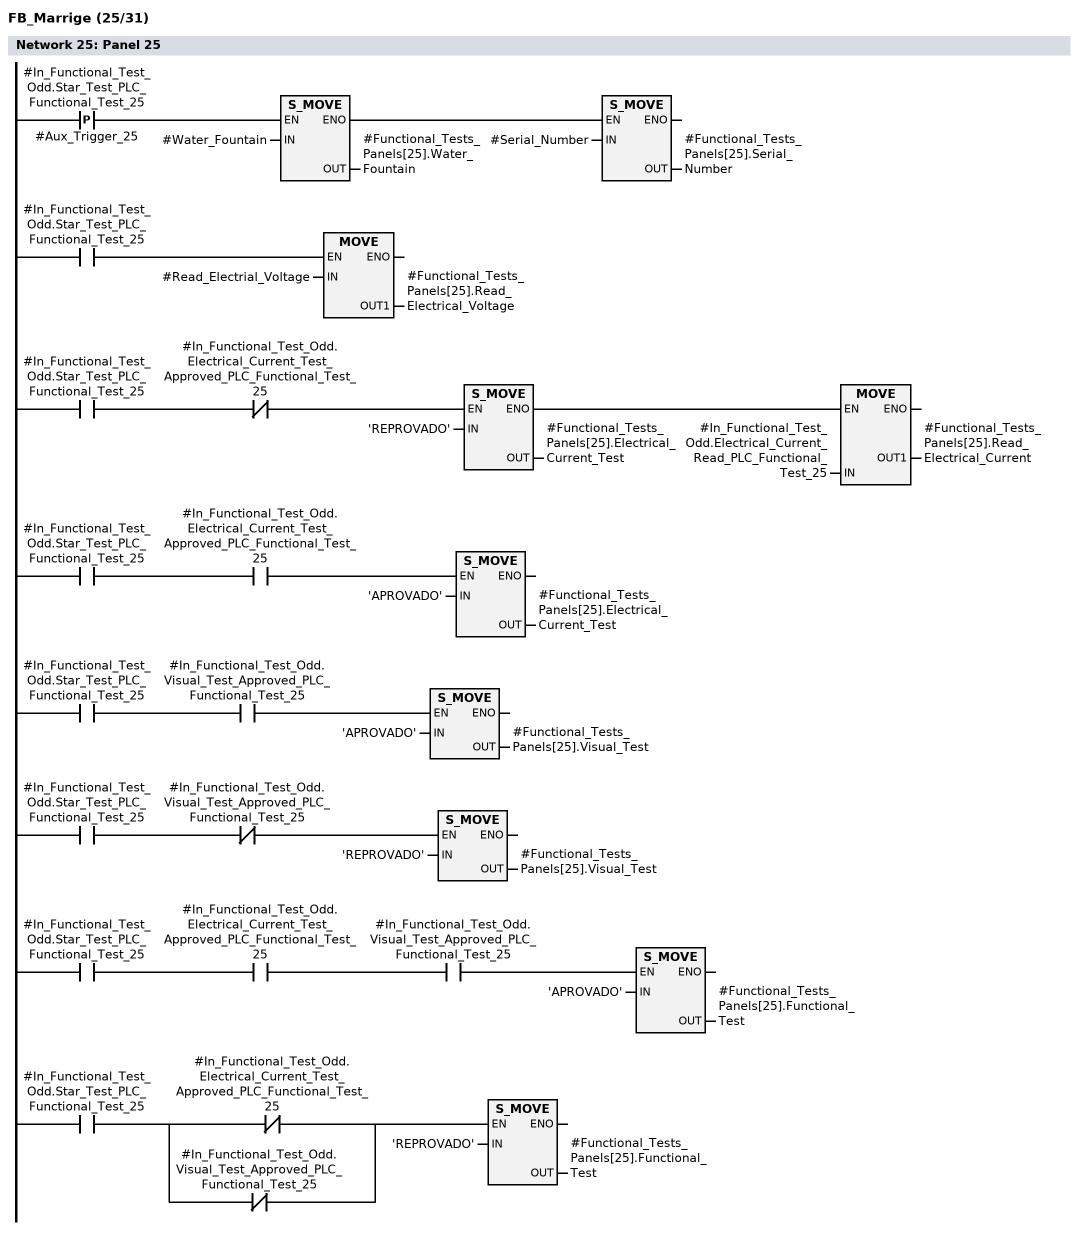
   RUNG wire#powerrail
      P_Contact(operand := #In_Functional_Test_Odd.Star_Test_PLC_Functional_Test_25, bit := #Aux_Trigger_25)
      S_Move(in := #Water_Fountain, out => #Functional_Tests_Panels[25].Water_Fountain)
      S_Move(in := #Serial_Number, out => #Functional_Tests_Panels[25].Serial_Number)
   END_RUNG
   RUNG wire#powerrail
      Contact( #In_Functional_Test_Odd.Star_Test_PLC_Functional_Test_25 )
      Move(in := #Read_Electrial_Voltage, out1 => #Functional_Tests_Panels[25].Read_Electrical_Voltage)
   END_RUNG
   RUNG wire#powerrail
      Contact( #In_Functional_Test_Odd.Star_Test_PLC_Functional_Test_25 )
      I_Contact( #In_Functional_Test_Odd.Electrical_Current_Test_Approved_PLC_Functional_Test_25 )
      S_Move(in := 'REPROVADO', out => #Functional_Tests_Panels[25].Electrical_Current_Test)
      Move(in := #In_Functional_Test_Odd.Electrical_Current_Read_PLC_Functional_Test_25, out1 => #Functional_Tests_Panels[25].Read_Electrical_Current)
   END_RUNG
   RUNG wire#powerrail
      Contact( #In_Functional_Test_Odd.Star_Test_PLC_Functional_Test_25 )
      Contact( #In_Functional_Test_Odd.Electrical_Current_Test_Approved_PLC_Functional_Test_25 )
      S_Move(in := 'APROVADO', out => #Functional_Tests_Panels[25].Electrical_Current_Test)
   END_RUNG
   RUNG wire#powerrail
      Contact( #In_Functional_Test_Odd.Star_Test_PLC_Functional_Test_25 )
      Contact( #In_Functional_Test_Odd.Visual_Test_Approved_PLC_Functional_Test_25 )
      S_Move(in := 'APROVADO', out => #Functional_Tests_Panels[25].Visual_Test)
   END_RUNG
   RUNG wire#powerrail
      Contact( #In_Functional_Test_Odd.Star_Test_PLC_Functional_Test_25 )
      I_Contact( #In_Functional_Test_Odd.Visual_Test_Approved_PLC_Functional_Test_25 )
      S_Move(in := 'REPROVADO', out => #Functional_Tests_Panels[25].Visual_Test)
   END_RUNG
   RUNG wire#powerrail
      Contact( #In_Functional_Test_Odd.Star_Test_PLC_Functional_Test_25 )
      Contact( #In_Functional_Test_Odd.Electrical_Current_Test_Approved_PLC_Functional_Test_25 )
      Contact( #In_Functional_Test_Odd.Visual_Test_Approved_PLC_Functional_Test_25 )
      S_Move(in := 'APROVADO', out => #Functional_Tests_Panels[25].Functional_Test)
   END_RUNG
   RUNG wire#powerrail
      Contact( #In_Functional_Test_Odd.Star_Test_PLC_Functional_Test_25 )
      wire#w1
      I_Contact( #In_Functional_Test_Odd.Electrical_Current_Test_Approved_PLC_Functional_Test_25 )
      wire#w2
      S_Move(in := 'REPROVADO', out => #Functional_Tests_Panels[25].Functional_Test)
   END_RUNG
   RUNG wire#w1
      I_Contact( #In_Functional_Test_Odd.Visual_Test_Approved_PLC_Functional_Test_25 )
   END_RUNG wire#w2
   // the same network as SCL:
   #_w1 := #In_Functional_Test_Odd.Star_Test_PLC_Functional_Test_25 AND NOT #Aux_Trigger_25;   // rising edge of #In_Functional_Test_Odd.Star_Test_PLC_Functional_Test_25
   #Aux_Trigger_25 := #In_Functional_Test_Odd.Star_Test_PLC_Functional_Test_25;
   IF #_w1 THEN
       #Functional_Tests_Panels[25].Water_Fountain := #Water_Fountain;
       #Functional_Tests_Panels[25].Serial_Number := #Serial_Number;
   END_IF;
   IF #In_Functional_Test_Odd.Star_Test_PLC_Functional_Test_25 THEN
       #Functional_Tests_Panels[25].Read_Electrical_Voltage := #Read_Electrial_Voltage;
   END_IF;
   IF #In_Functional_Test_Odd.Star_Test_PLC_Functional_Test_25 AND NOT #In_Functional_Test_Odd.Electrical_Current_Test_Approved_PLC_Functional_Test_25 THEN
       #Functional_Tests_Panels[25].Electrical_Current_Test := 'REPROVADO';
       #Functional_Tests_Panels[25].Read_Electrical_Current := #In_Functional_Test_Odd.Electrical_Current_Read_PLC_Functional_Test_25;
   END_IF;
   IF #In_Functional_Test_Odd.Star_Test_PLC_Functional_Test_25 AND #In_Functional_Test_Odd.Electrical_Current_Test_Approved_PLC_Functional_Test_25 THEN
       #Functional_Tests_Panels[25].Electrical_Current_Test := 'APROVADO';
   END_IF;
   IF #In_Functional_Test_Odd.Star_Test_PLC_Functional_Test_25 AND #In_Functional_Test_Odd.Visual_Test_Approved_PLC_Functional_Test_25 THEN
       #Functional_Tests_Panels[25].Visual_Test := 'APROVADO';
   END_IF;
   IF #In_Functional_Test_Odd.Star_Test_PLC_Functional_Test_25 AND NOT #In_Functional_Test_Odd.Visual_Test_Approved_PLC_Functional_Test_25 THEN
       #Functional_Tests_Panels[25].Visual_Test := 'REPROVADO';
   END_IF;
   IF #In_Functional_Test_Odd.Star_Test_PLC_Functional_Test_25 AND #In_Functional_Test_Odd.Electrical_Current_Test_Approved_PLC_Functional_Test_25 AND #In_Functional_Test_Odd.Visual_Test_Approved_PLC_Functional_Test_25 THEN
       #Functional_Tests_Panels[25].Functional_Test := 'APROVADO';
   END_IF;
   IF #In_Functional_Test_Odd.Star_Test_PLC_Functional_Test_25 AND (NOT #In_Functional_Test_Odd.Electrical_Current_Test_Approved_PLC_Functional_Test_25 OR NOT #In_Functional_Test_Odd.Visual_Test_Approved_PLC_Functional_Test_25) THEN
       #Functional_Tests_Panels[25].Functional_Test := 'REPROVADO';
   END_IF;
END_REGION

REGION Network 26: Panel 26
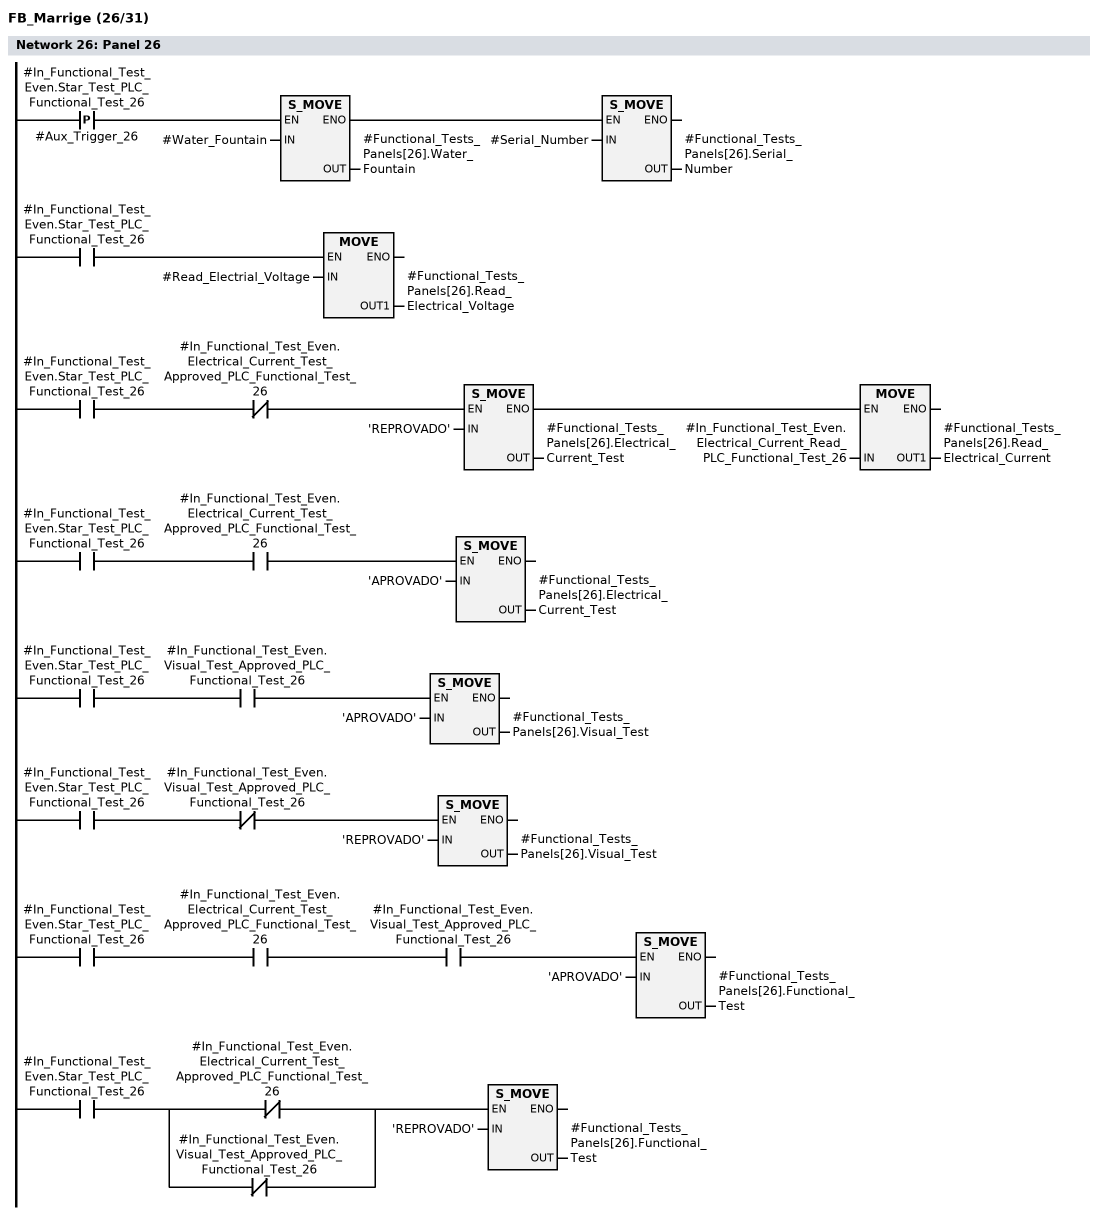
   RUNG wire#powerrail
      P_Contact(operand := #In_Functional_Test_Even.Star_Test_PLC_Functional_Test_26, bit := #Aux_Trigger_26)
      S_Move(in := #Water_Fountain, out => #Functional_Tests_Panels[26].Water_Fountain)
      S_Move(in := #Serial_Number, out => #Functional_Tests_Panels[26].Serial_Number)
   END_RUNG
   RUNG wire#powerrail
      Contact( #In_Functional_Test_Even.Star_Test_PLC_Functional_Test_26 )
      Move(in := #Read_Electrial_Voltage, out1 => #Functional_Tests_Panels[26].Read_Electrical_Voltage)
   END_RUNG
   RUNG wire#powerrail
      Contact( #In_Functional_Test_Even.Star_Test_PLC_Functional_Test_26 )
      I_Contact( #In_Functional_Test_Even.Electrical_Current_Test_Approved_PLC_Functional_Test_26 )
      S_Move(in := 'REPROVADO', out => #Functional_Tests_Panels[26].Electrical_Current_Test)
      Move(in := #In_Functional_Test_Even.Electrical_Current_Read_PLC_Functional_Test_26, out1 => #Functional_Tests_Panels[26].Read_Electrical_Current)
   END_RUNG
   RUNG wire#powerrail
      Contact( #In_Functional_Test_Even.Star_Test_PLC_Functional_Test_26 )
      Contact( #In_Functional_Test_Even.Electrical_Current_Test_Approved_PLC_Functional_Test_26 )
      S_Move(in := 'APROVADO', out => #Functional_Tests_Panels[26].Electrical_Current_Test)
   END_RUNG
   RUNG wire#powerrail
      Contact( #In_Functional_Test_Even.Star_Test_PLC_Functional_Test_26 )
      Contact( #In_Functional_Test_Even.Visual_Test_Approved_PLC_Functional_Test_26 )
      S_Move(in := 'APROVADO', out => #Functional_Tests_Panels[26].Visual_Test)
   END_RUNG
   RUNG wire#powerrail
      Contact( #In_Functional_Test_Even.Star_Test_PLC_Functional_Test_26 )
      I_Contact( #In_Functional_Test_Even.Visual_Test_Approved_PLC_Functional_Test_26 )
      S_Move(in := 'REPROVADO', out => #Functional_Tests_Panels[26].Visual_Test)
   END_RUNG
   RUNG wire#powerrail
      Contact( #In_Functional_Test_Even.Star_Test_PLC_Functional_Test_26 )
      Contact( #In_Functional_Test_Even.Electrical_Current_Test_Approved_PLC_Functional_Test_26 )
      Contact( #In_Functional_Test_Even.Visual_Test_Approved_PLC_Functional_Test_26 )
      S_Move(in := 'APROVADO', out => #Functional_Tests_Panels[26].Functional_Test)
   END_RUNG
   RUNG wire#powerrail
      Contact( #In_Functional_Test_Even.Star_Test_PLC_Functional_Test_26 )
      wire#w1
      I_Contact( #In_Functional_Test_Even.Electrical_Current_Test_Approved_PLC_Functional_Test_26 )
      wire#w2
      S_Move(in := 'REPROVADO', out => #Functional_Tests_Panels[26].Functional_Test)
   END_RUNG
   RUNG wire#w1
      I_Contact( #In_Functional_Test_Even.Visual_Test_Approved_PLC_Functional_Test_26 )
   END_RUNG wire#w2
   // the same network as SCL:
   #_w1 := #In_Functional_Test_Even.Star_Test_PLC_Functional_Test_26 AND NOT #Aux_Trigger_26;   // rising edge of #In_Functional_Test_Even.Star_Test_PLC_Functional_Test_26
   #Aux_Trigger_26 := #In_Functional_Test_Even.Star_Test_PLC_Functional_Test_26;
   IF #_w1 THEN
       #Functional_Tests_Panels[26].Water_Fountain := #Water_Fountain;
       #Functional_Tests_Panels[26].Serial_Number := #Serial_Number;
   END_IF;
   IF #In_Functional_Test_Even.Star_Test_PLC_Functional_Test_26 THEN
       #Functional_Tests_Panels[26].Read_Electrical_Voltage := #Read_Electrial_Voltage;
   END_IF;
   IF #In_Functional_Test_Even.Star_Test_PLC_Functional_Test_26 AND NOT #In_Functional_Test_Even.Electrical_Current_Test_Approved_PLC_Functional_Test_26 THEN
       #Functional_Tests_Panels[26].Electrical_Current_Test := 'REPROVADO';
       #Functional_Tests_Panels[26].Read_Electrical_Current := #In_Functional_Test_Even.Electrical_Current_Read_PLC_Functional_Test_26;
   END_IF;
   IF #In_Functional_Test_Even.Star_Test_PLC_Functional_Test_26 AND #In_Functional_Test_Even.Electrical_Current_Test_Approved_PLC_Functional_Test_26 THEN
       #Functional_Tests_Panels[26].Electrical_Current_Test := 'APROVADO';
   END_IF;
   IF #In_Functional_Test_Even.Star_Test_PLC_Functional_Test_26 AND #In_Functional_Test_Even.Visual_Test_Approved_PLC_Functional_Test_26 THEN
       #Functional_Tests_Panels[26].Visual_Test := 'APROVADO';
   END_IF;
   IF #In_Functional_Test_Even.Star_Test_PLC_Functional_Test_26 AND NOT #In_Functional_Test_Even.Visual_Test_Approved_PLC_Functional_Test_26 THEN
       #Functional_Tests_Panels[26].Visual_Test := 'REPROVADO';
   END_IF;
   IF #In_Functional_Test_Even.Star_Test_PLC_Functional_Test_26 AND #In_Functional_Test_Even.Electrical_Current_Test_Approved_PLC_Functional_Test_26 AND #In_Functional_Test_Even.Visual_Test_Approved_PLC_Functional_Test_26 THEN
       #Functional_Tests_Panels[26].Functional_Test := 'APROVADO';
   END_IF;
   IF #In_Functional_Test_Even.Star_Test_PLC_Functional_Test_26 AND (NOT #In_Functional_Test_Even.Electrical_Current_Test_Approved_PLC_Functional_Test_26 OR NOT #In_Functional_Test_Even.Visual_Test_Approved_PLC_Functional_Test_26) THEN
       #Functional_Tests_Panels[26].Functional_Test := 'REPROVADO';
   END_IF;
END_REGION

REGION Network 27: Panel 27
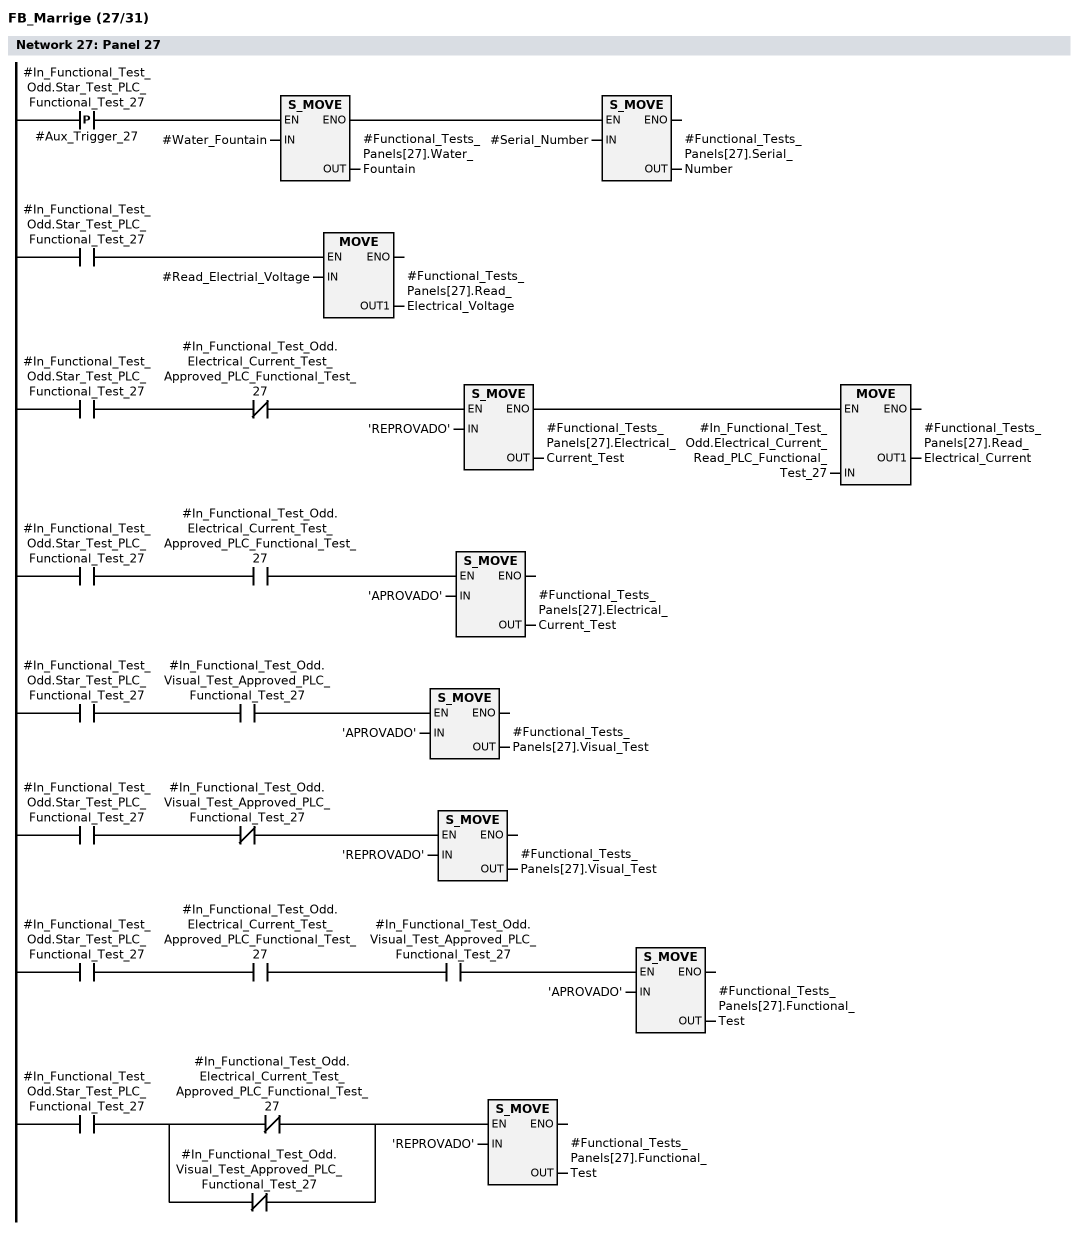
   RUNG wire#powerrail
      P_Contact(operand := #In_Functional_Test_Odd.Star_Test_PLC_Functional_Test_27, bit := #Aux_Trigger_27)
      S_Move(in := #Water_Fountain, out => #Functional_Tests_Panels[27].Water_Fountain)
      S_Move(in := #Serial_Number, out => #Functional_Tests_Panels[27].Serial_Number)
   END_RUNG
   RUNG wire#powerrail
      Contact( #In_Functional_Test_Odd.Star_Test_PLC_Functional_Test_27 )
      Move(in := #Read_Electrial_Voltage, out1 => #Functional_Tests_Panels[27].Read_Electrical_Voltage)
   END_RUNG
   RUNG wire#powerrail
      Contact( #In_Functional_Test_Odd.Star_Test_PLC_Functional_Test_27 )
      I_Contact( #In_Functional_Test_Odd.Electrical_Current_Test_Approved_PLC_Functional_Test_27 )
      S_Move(in := 'REPROVADO', out => #Functional_Tests_Panels[27].Electrical_Current_Test)
      Move(in := #In_Functional_Test_Odd.Electrical_Current_Read_PLC_Functional_Test_27, out1 => #Functional_Tests_Panels[27].Read_Electrical_Current)
   END_RUNG
   RUNG wire#powerrail
      Contact( #In_Functional_Test_Odd.Star_Test_PLC_Functional_Test_27 )
      Contact( #In_Functional_Test_Odd.Electrical_Current_Test_Approved_PLC_Functional_Test_27 )
      S_Move(in := 'APROVADO', out => #Functional_Tests_Panels[27].Electrical_Current_Test)
   END_RUNG
   RUNG wire#powerrail
      Contact( #In_Functional_Test_Odd.Star_Test_PLC_Functional_Test_27 )
      Contact( #In_Functional_Test_Odd.Visual_Test_Approved_PLC_Functional_Test_27 )
      S_Move(in := 'APROVADO', out => #Functional_Tests_Panels[27].Visual_Test)
   END_RUNG
   RUNG wire#powerrail
      Contact( #In_Functional_Test_Odd.Star_Test_PLC_Functional_Test_27 )
      I_Contact( #In_Functional_Test_Odd.Visual_Test_Approved_PLC_Functional_Test_27 )
      S_Move(in := 'REPROVADO', out => #Functional_Tests_Panels[27].Visual_Test)
   END_RUNG
   RUNG wire#powerrail
      Contact( #In_Functional_Test_Odd.Star_Test_PLC_Functional_Test_27 )
      Contact( #In_Functional_Test_Odd.Electrical_Current_Test_Approved_PLC_Functional_Test_27 )
      Contact( #In_Functional_Test_Odd.Visual_Test_Approved_PLC_Functional_Test_27 )
      S_Move(in := 'APROVADO', out => #Functional_Tests_Panels[27].Functional_Test)
   END_RUNG
   RUNG wire#powerrail
      Contact( #In_Functional_Test_Odd.Star_Test_PLC_Functional_Test_27 )
      wire#w1
      I_Contact( #In_Functional_Test_Odd.Electrical_Current_Test_Approved_PLC_Functional_Test_27 )
      wire#w2
      S_Move(in := 'REPROVADO', out => #Functional_Tests_Panels[27].Functional_Test)
   END_RUNG
   RUNG wire#w1
      I_Contact( #In_Functional_Test_Odd.Visual_Test_Approved_PLC_Functional_Test_27 )
   END_RUNG wire#w2
   // the same network as SCL:
   #_w1 := #In_Functional_Test_Odd.Star_Test_PLC_Functional_Test_27 AND NOT #Aux_Trigger_27;   // rising edge of #In_Functional_Test_Odd.Star_Test_PLC_Functional_Test_27
   #Aux_Trigger_27 := #In_Functional_Test_Odd.Star_Test_PLC_Functional_Test_27;
   IF #_w1 THEN
       #Functional_Tests_Panels[27].Water_Fountain := #Water_Fountain;
       #Functional_Tests_Panels[27].Serial_Number := #Serial_Number;
   END_IF;
   IF #In_Functional_Test_Odd.Star_Test_PLC_Functional_Test_27 THEN
       #Functional_Tests_Panels[27].Read_Electrical_Voltage := #Read_Electrial_Voltage;
   END_IF;
   IF #In_Functional_Test_Odd.Star_Test_PLC_Functional_Test_27 AND NOT #In_Functional_Test_Odd.Electrical_Current_Test_Approved_PLC_Functional_Test_27 THEN
       #Functional_Tests_Panels[27].Electrical_Current_Test := 'REPROVADO';
       #Functional_Tests_Panels[27].Read_Electrical_Current := #In_Functional_Test_Odd.Electrical_Current_Read_PLC_Functional_Test_27;
   END_IF;
   IF #In_Functional_Test_Odd.Star_Test_PLC_Functional_Test_27 AND #In_Functional_Test_Odd.Electrical_Current_Test_Approved_PLC_Functional_Test_27 THEN
       #Functional_Tests_Panels[27].Electrical_Current_Test := 'APROVADO';
   END_IF;
   IF #In_Functional_Test_Odd.Star_Test_PLC_Functional_Test_27 AND #In_Functional_Test_Odd.Visual_Test_Approved_PLC_Functional_Test_27 THEN
       #Functional_Tests_Panels[27].Visual_Test := 'APROVADO';
   END_IF;
   IF #In_Functional_Test_Odd.Star_Test_PLC_Functional_Test_27 AND NOT #In_Functional_Test_Odd.Visual_Test_Approved_PLC_Functional_Test_27 THEN
       #Functional_Tests_Panels[27].Visual_Test := 'REPROVADO';
   END_IF;
   IF #In_Functional_Test_Odd.Star_Test_PLC_Functional_Test_27 AND #In_Functional_Test_Odd.Electrical_Current_Test_Approved_PLC_Functional_Test_27 AND #In_Functional_Test_Odd.Visual_Test_Approved_PLC_Functional_Test_27 THEN
       #Functional_Tests_Panels[27].Functional_Test := 'APROVADO';
   END_IF;
   IF #In_Functional_Test_Odd.Star_Test_PLC_Functional_Test_27 AND (NOT #In_Functional_Test_Odd.Electrical_Current_Test_Approved_PLC_Functional_Test_27 OR NOT #In_Functional_Test_Odd.Visual_Test_Approved_PLC_Functional_Test_27) THEN
       #Functional_Tests_Panels[27].Functional_Test := 'REPROVADO';
   END_IF;
END_REGION

REGION Network 28: Panel 28
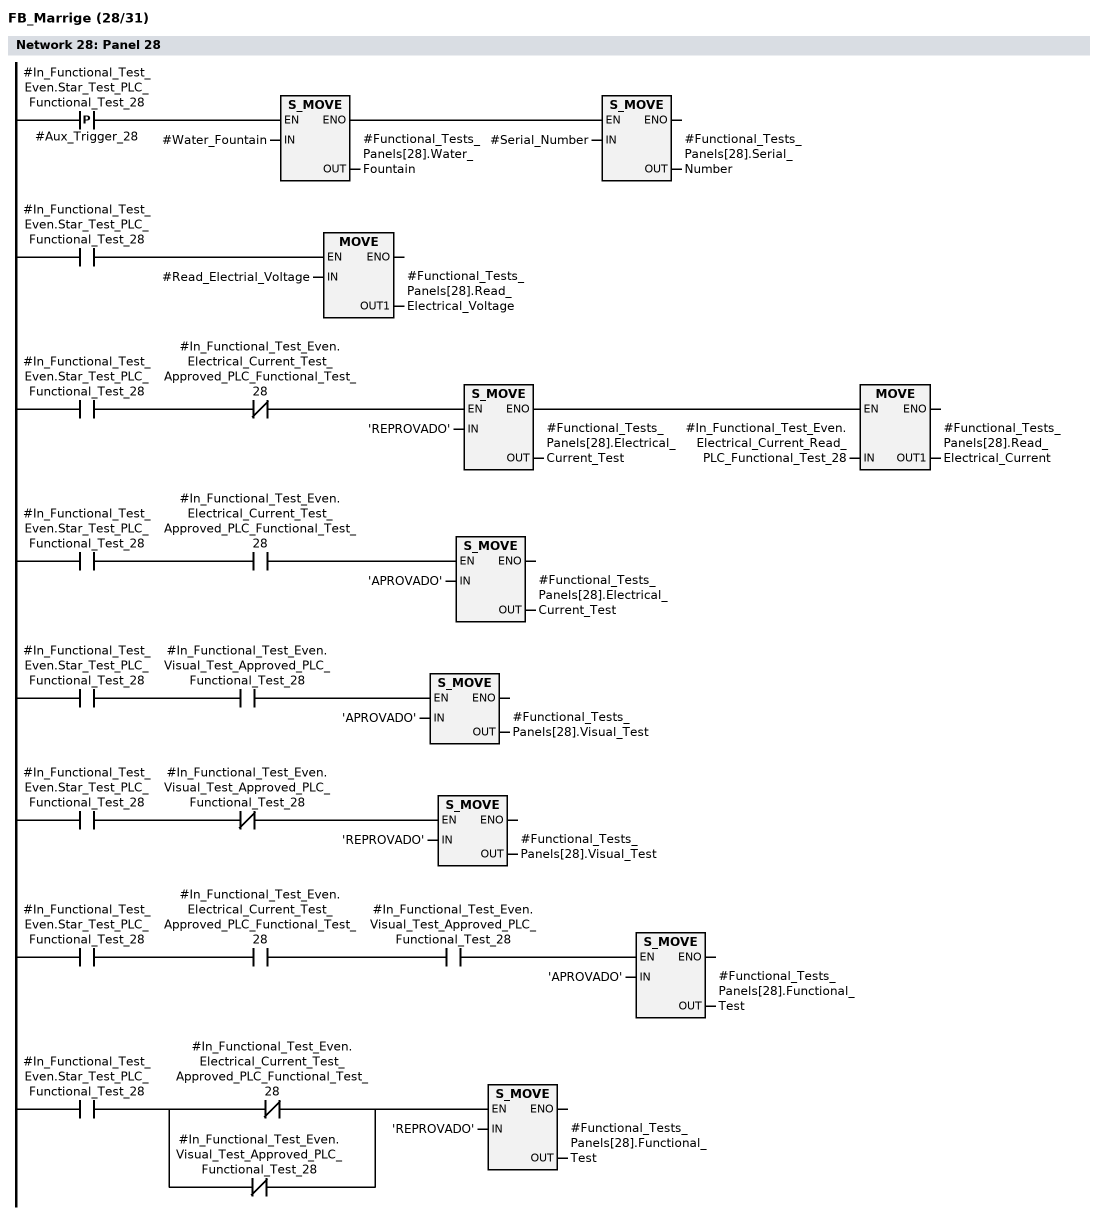
   RUNG wire#powerrail
      P_Contact(operand := #In_Functional_Test_Even.Star_Test_PLC_Functional_Test_28, bit := #Aux_Trigger_28)
      S_Move(in := #Water_Fountain, out => #Functional_Tests_Panels[28].Water_Fountain)
      S_Move(in := #Serial_Number, out => #Functional_Tests_Panels[28].Serial_Number)
   END_RUNG
   RUNG wire#powerrail
      Contact( #In_Functional_Test_Even.Star_Test_PLC_Functional_Test_28 )
      Move(in := #Read_Electrial_Voltage, out1 => #Functional_Tests_Panels[28].Read_Electrical_Voltage)
   END_RUNG
   RUNG wire#powerrail
      Contact( #In_Functional_Test_Even.Star_Test_PLC_Functional_Test_28 )
      I_Contact( #In_Functional_Test_Even.Electrical_Current_Test_Approved_PLC_Functional_Test_28 )
      S_Move(in := 'REPROVADO', out => #Functional_Tests_Panels[28].Electrical_Current_Test)
      Move(in := #In_Functional_Test_Even.Electrical_Current_Read_PLC_Functional_Test_28, out1 => #Functional_Tests_Panels[28].Read_Electrical_Current)
   END_RUNG
   RUNG wire#powerrail
      Contact( #In_Functional_Test_Even.Star_Test_PLC_Functional_Test_28 )
      Contact( #In_Functional_Test_Even.Electrical_Current_Test_Approved_PLC_Functional_Test_28 )
      S_Move(in := 'APROVADO', out => #Functional_Tests_Panels[28].Electrical_Current_Test)
   END_RUNG
   RUNG wire#powerrail
      Contact( #In_Functional_Test_Even.Star_Test_PLC_Functional_Test_28 )
      Contact( #In_Functional_Test_Even.Visual_Test_Approved_PLC_Functional_Test_28 )
      S_Move(in := 'APROVADO', out => #Functional_Tests_Panels[28].Visual_Test)
   END_RUNG
   RUNG wire#powerrail
      Contact( #In_Functional_Test_Even.Star_Test_PLC_Functional_Test_28 )
      I_Contact( #In_Functional_Test_Even.Visual_Test_Approved_PLC_Functional_Test_28 )
      S_Move(in := 'REPROVADO', out => #Functional_Tests_Panels[28].Visual_Test)
   END_RUNG
   RUNG wire#powerrail
      Contact( #In_Functional_Test_Even.Star_Test_PLC_Functional_Test_28 )
      Contact( #In_Functional_Test_Even.Electrical_Current_Test_Approved_PLC_Functional_Test_28 )
      Contact( #In_Functional_Test_Even.Visual_Test_Approved_PLC_Functional_Test_28 )
      S_Move(in := 'APROVADO', out => #Functional_Tests_Panels[28].Functional_Test)
   END_RUNG
   RUNG wire#powerrail
      Contact( #In_Functional_Test_Even.Star_Test_PLC_Functional_Test_28 )
      wire#w1
      I_Contact( #In_Functional_Test_Even.Electrical_Current_Test_Approved_PLC_Functional_Test_28 )
      wire#w2
      S_Move(in := 'REPROVADO', out => #Functional_Tests_Panels[28].Functional_Test)
   END_RUNG
   RUNG wire#w1
      I_Contact( #In_Functional_Test_Even.Visual_Test_Approved_PLC_Functional_Test_28 )
   END_RUNG wire#w2
   // the same network as SCL:
   #_w1 := #In_Functional_Test_Even.Star_Test_PLC_Functional_Test_28 AND NOT #Aux_Trigger_28;   // rising edge of #In_Functional_Test_Even.Star_Test_PLC_Functional_Test_28
   #Aux_Trigger_28 := #In_Functional_Test_Even.Star_Test_PLC_Functional_Test_28;
   IF #_w1 THEN
       #Functional_Tests_Panels[28].Water_Fountain := #Water_Fountain;
       #Functional_Tests_Panels[28].Serial_Number := #Serial_Number;
   END_IF;
   IF #In_Functional_Test_Even.Star_Test_PLC_Functional_Test_28 THEN
       #Functional_Tests_Panels[28].Read_Electrical_Voltage := #Read_Electrial_Voltage;
   END_IF;
   IF #In_Functional_Test_Even.Star_Test_PLC_Functional_Test_28 AND NOT #In_Functional_Test_Even.Electrical_Current_Test_Approved_PLC_Functional_Test_28 THEN
       #Functional_Tests_Panels[28].Electrical_Current_Test := 'REPROVADO';
       #Functional_Tests_Panels[28].Read_Electrical_Current := #In_Functional_Test_Even.Electrical_Current_Read_PLC_Functional_Test_28;
   END_IF;
   IF #In_Functional_Test_Even.Star_Test_PLC_Functional_Test_28 AND #In_Functional_Test_Even.Electrical_Current_Test_Approved_PLC_Functional_Test_28 THEN
       #Functional_Tests_Panels[28].Electrical_Current_Test := 'APROVADO';
   END_IF;
   IF #In_Functional_Test_Even.Star_Test_PLC_Functional_Test_28 AND #In_Functional_Test_Even.Visual_Test_Approved_PLC_Functional_Test_28 THEN
       #Functional_Tests_Panels[28].Visual_Test := 'APROVADO';
   END_IF;
   IF #In_Functional_Test_Even.Star_Test_PLC_Functional_Test_28 AND NOT #In_Functional_Test_Even.Visual_Test_Approved_PLC_Functional_Test_28 THEN
       #Functional_Tests_Panels[28].Visual_Test := 'REPROVADO';
   END_IF;
   IF #In_Functional_Test_Even.Star_Test_PLC_Functional_Test_28 AND #In_Functional_Test_Even.Electrical_Current_Test_Approved_PLC_Functional_Test_28 AND #In_Functional_Test_Even.Visual_Test_Approved_PLC_Functional_Test_28 THEN
       #Functional_Tests_Panels[28].Functional_Test := 'APROVADO';
   END_IF;
   IF #In_Functional_Test_Even.Star_Test_PLC_Functional_Test_28 AND (NOT #In_Functional_Test_Even.Electrical_Current_Test_Approved_PLC_Functional_Test_28 OR NOT #In_Functional_Test_Even.Visual_Test_Approved_PLC_Functional_Test_28) THEN
       #Functional_Tests_Panels[28].Functional_Test := 'REPROVADO';
   END_IF;
END_REGION

REGION Network 29: Panel 29
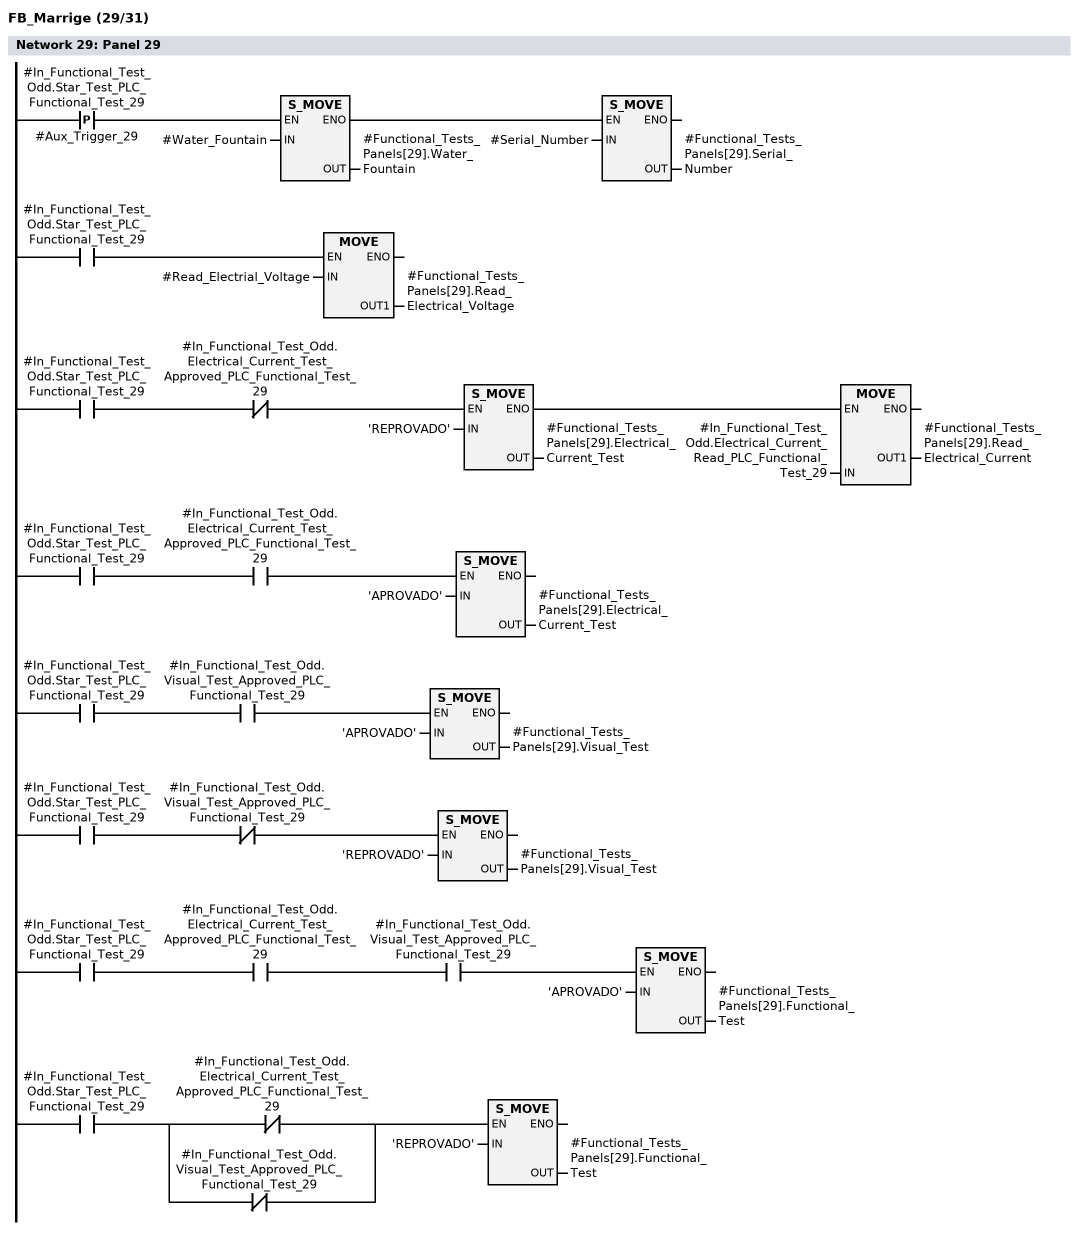
   RUNG wire#powerrail
      P_Contact(operand := #In_Functional_Test_Odd.Star_Test_PLC_Functional_Test_29, bit := #Aux_Trigger_29)
      S_Move(in := #Water_Fountain, out => #Functional_Tests_Panels[29].Water_Fountain)
      S_Move(in := #Serial_Number, out => #Functional_Tests_Panels[29].Serial_Number)
   END_RUNG
   RUNG wire#powerrail
      Contact( #In_Functional_Test_Odd.Star_Test_PLC_Functional_Test_29 )
      Move(in := #Read_Electrial_Voltage, out1 => #Functional_Tests_Panels[29].Read_Electrical_Voltage)
   END_RUNG
   RUNG wire#powerrail
      Contact( #In_Functional_Test_Odd.Star_Test_PLC_Functional_Test_29 )
      I_Contact( #In_Functional_Test_Odd.Electrical_Current_Test_Approved_PLC_Functional_Test_29 )
      S_Move(in := 'REPROVADO', out => #Functional_Tests_Panels[29].Electrical_Current_Test)
      Move(in := #In_Functional_Test_Odd.Electrical_Current_Read_PLC_Functional_Test_29, out1 => #Functional_Tests_Panels[29].Read_Electrical_Current)
   END_RUNG
   RUNG wire#powerrail
      Contact( #In_Functional_Test_Odd.Star_Test_PLC_Functional_Test_29 )
      Contact( #In_Functional_Test_Odd.Electrical_Current_Test_Approved_PLC_Functional_Test_29 )
      S_Move(in := 'APROVADO', out => #Functional_Tests_Panels[29].Electrical_Current_Test)
   END_RUNG
   RUNG wire#powerrail
      Contact( #In_Functional_Test_Odd.Star_Test_PLC_Functional_Test_29 )
      Contact( #In_Functional_Test_Odd.Visual_Test_Approved_PLC_Functional_Test_29 )
      S_Move(in := 'APROVADO', out => #Functional_Tests_Panels[29].Visual_Test)
   END_RUNG
   RUNG wire#powerrail
      Contact( #In_Functional_Test_Odd.Star_Test_PLC_Functional_Test_29 )
      I_Contact( #In_Functional_Test_Odd.Visual_Test_Approved_PLC_Functional_Test_29 )
      S_Move(in := 'REPROVADO', out => #Functional_Tests_Panels[29].Visual_Test)
   END_RUNG
   RUNG wire#powerrail
      Contact( #In_Functional_Test_Odd.Star_Test_PLC_Functional_Test_29 )
      Contact( #In_Functional_Test_Odd.Electrical_Current_Test_Approved_PLC_Functional_Test_29 )
      Contact( #In_Functional_Test_Odd.Visual_Test_Approved_PLC_Functional_Test_29 )
      S_Move(in := 'APROVADO', out => #Functional_Tests_Panels[29].Functional_Test)
   END_RUNG
   RUNG wire#powerrail
      Contact( #In_Functional_Test_Odd.Star_Test_PLC_Functional_Test_29 )
      wire#w1
      I_Contact( #In_Functional_Test_Odd.Electrical_Current_Test_Approved_PLC_Functional_Test_29 )
      wire#w2
      S_Move(in := 'REPROVADO', out => #Functional_Tests_Panels[29].Functional_Test)
   END_RUNG
   RUNG wire#w1
      I_Contact( #In_Functional_Test_Odd.Visual_Test_Approved_PLC_Functional_Test_29 )
   END_RUNG wire#w2
   // the same network as SCL:
   #_w1 := #In_Functional_Test_Odd.Star_Test_PLC_Functional_Test_29 AND NOT #Aux_Trigger_29;   // rising edge of #In_Functional_Test_Odd.Star_Test_PLC_Functional_Test_29
   #Aux_Trigger_29 := #In_Functional_Test_Odd.Star_Test_PLC_Functional_Test_29;
   IF #_w1 THEN
       #Functional_Tests_Panels[29].Water_Fountain := #Water_Fountain;
       #Functional_Tests_Panels[29].Serial_Number := #Serial_Number;
   END_IF;
   IF #In_Functional_Test_Odd.Star_Test_PLC_Functional_Test_29 THEN
       #Functional_Tests_Panels[29].Read_Electrical_Voltage := #Read_Electrial_Voltage;
   END_IF;
   IF #In_Functional_Test_Odd.Star_Test_PLC_Functional_Test_29 AND NOT #In_Functional_Test_Odd.Electrical_Current_Test_Approved_PLC_Functional_Test_29 THEN
       #Functional_Tests_Panels[29].Electrical_Current_Test := 'REPROVADO';
       #Functional_Tests_Panels[29].Read_Electrical_Current := #In_Functional_Test_Odd.Electrical_Current_Read_PLC_Functional_Test_29;
   END_IF;
   IF #In_Functional_Test_Odd.Star_Test_PLC_Functional_Test_29 AND #In_Functional_Test_Odd.Electrical_Current_Test_Approved_PLC_Functional_Test_29 THEN
       #Functional_Tests_Panels[29].Electrical_Current_Test := 'APROVADO';
   END_IF;
   IF #In_Functional_Test_Odd.Star_Test_PLC_Functional_Test_29 AND #In_Functional_Test_Odd.Visual_Test_Approved_PLC_Functional_Test_29 THEN
       #Functional_Tests_Panels[29].Visual_Test := 'APROVADO';
   END_IF;
   IF #In_Functional_Test_Odd.Star_Test_PLC_Functional_Test_29 AND NOT #In_Functional_Test_Odd.Visual_Test_Approved_PLC_Functional_Test_29 THEN
       #Functional_Tests_Panels[29].Visual_Test := 'REPROVADO';
   END_IF;
   IF #In_Functional_Test_Odd.Star_Test_PLC_Functional_Test_29 AND #In_Functional_Test_Odd.Electrical_Current_Test_Approved_PLC_Functional_Test_29 AND #In_Functional_Test_Odd.Visual_Test_Approved_PLC_Functional_Test_29 THEN
       #Functional_Tests_Panels[29].Functional_Test := 'APROVADO';
   END_IF;
   IF #In_Functional_Test_Odd.Star_Test_PLC_Functional_Test_29 AND (NOT #In_Functional_Test_Odd.Electrical_Current_Test_Approved_PLC_Functional_Test_29 OR NOT #In_Functional_Test_Odd.Visual_Test_Approved_PLC_Functional_Test_29) THEN
       #Functional_Tests_Panels[29].Functional_Test := 'REPROVADO';
   END_IF;
END_REGION

REGION Network 30: Panel 30
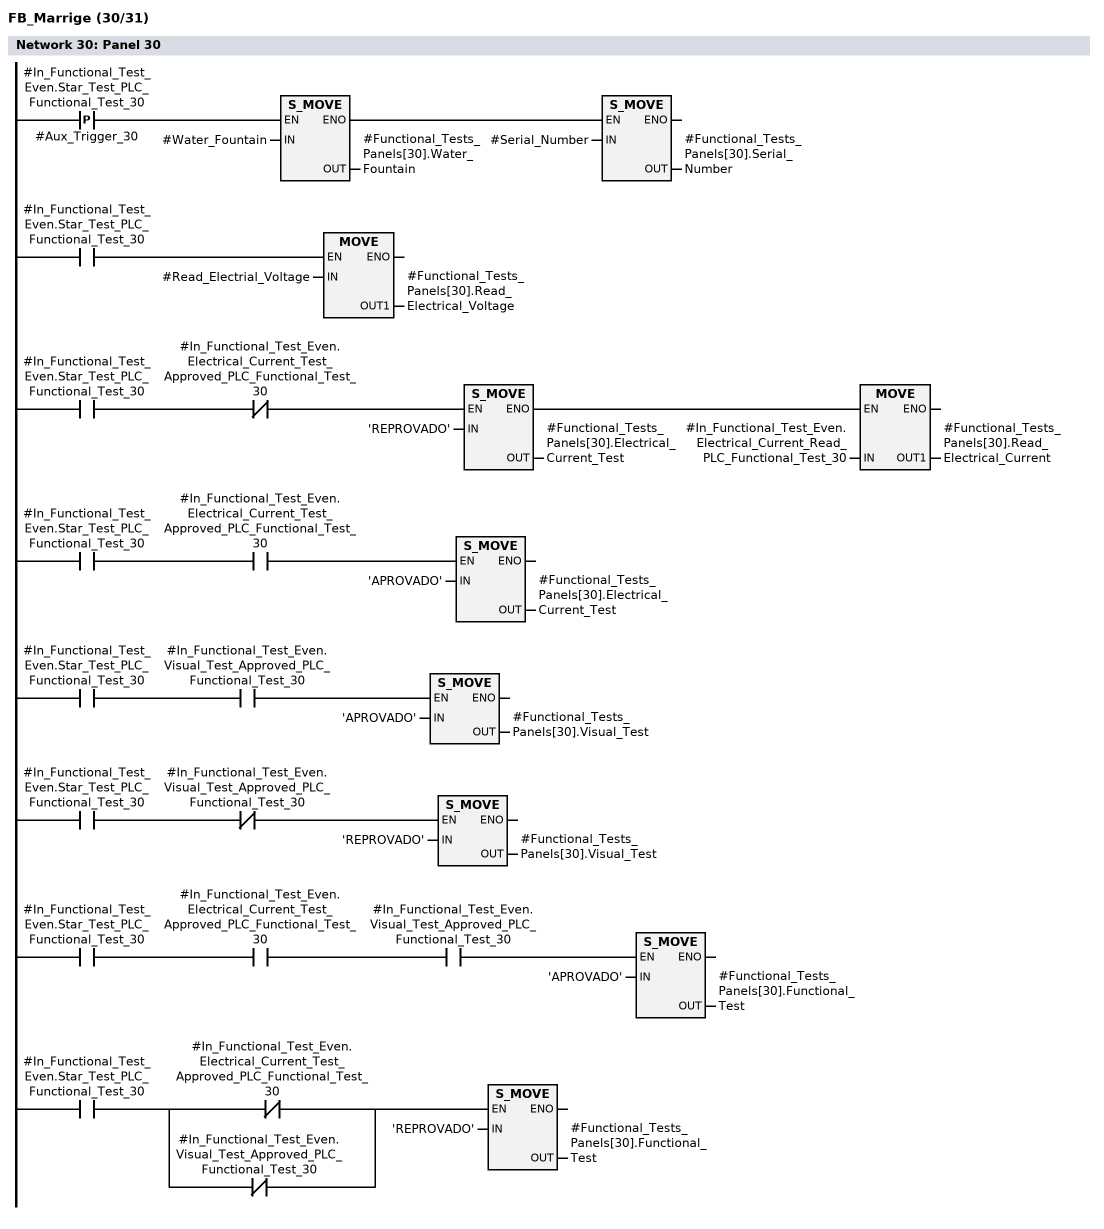
   RUNG wire#powerrail
      P_Contact(operand := #In_Functional_Test_Even.Star_Test_PLC_Functional_Test_30, bit := #Aux_Trigger_30)
      S_Move(in := #Water_Fountain, out => #Functional_Tests_Panels[30].Water_Fountain)
      S_Move(in := #Serial_Number, out => #Functional_Tests_Panels[30].Serial_Number)
   END_RUNG
   RUNG wire#powerrail
      Contact( #In_Functional_Test_Even.Star_Test_PLC_Functional_Test_30 )
      Move(in := #Read_Electrial_Voltage, out1 => #Functional_Tests_Panels[30].Read_Electrical_Voltage)
   END_RUNG
   RUNG wire#powerrail
      Contact( #In_Functional_Test_Even.Star_Test_PLC_Functional_Test_30 )
      I_Contact( #In_Functional_Test_Even.Electrical_Current_Test_Approved_PLC_Functional_Test_30 )
      S_Move(in := 'REPROVADO', out => #Functional_Tests_Panels[30].Electrical_Current_Test)
      Move(in := #In_Functional_Test_Even.Electrical_Current_Read_PLC_Functional_Test_30, out1 => #Functional_Tests_Panels[30].Read_Electrical_Current)
   END_RUNG
   RUNG wire#powerrail
      Contact( #In_Functional_Test_Even.Star_Test_PLC_Functional_Test_30 )
      Contact( #In_Functional_Test_Even.Electrical_Current_Test_Approved_PLC_Functional_Test_30 )
      S_Move(in := 'APROVADO', out => #Functional_Tests_Panels[30].Electrical_Current_Test)
   END_RUNG
   RUNG wire#powerrail
      Contact( #In_Functional_Test_Even.Star_Test_PLC_Functional_Test_30 )
      Contact( #In_Functional_Test_Even.Visual_Test_Approved_PLC_Functional_Test_30 )
      S_Move(in := 'APROVADO', out => #Functional_Tests_Panels[30].Visual_Test)
   END_RUNG
   RUNG wire#powerrail
      Contact( #In_Functional_Test_Even.Star_Test_PLC_Functional_Test_30 )
      I_Contact( #In_Functional_Test_Even.Visual_Test_Approved_PLC_Functional_Test_30 )
      S_Move(in := 'REPROVADO', out => #Functional_Tests_Panels[30].Visual_Test)
   END_RUNG
   RUNG wire#powerrail
      Contact( #In_Functional_Test_Even.Star_Test_PLC_Functional_Test_30 )
      Contact( #In_Functional_Test_Even.Electrical_Current_Test_Approved_PLC_Functional_Test_30 )
      Contact( #In_Functional_Test_Even.Visual_Test_Approved_PLC_Functional_Test_30 )
      S_Move(in := 'APROVADO', out => #Functional_Tests_Panels[30].Functional_Test)
   END_RUNG
   RUNG wire#powerrail
      Contact( #In_Functional_Test_Even.Star_Test_PLC_Functional_Test_30 )
      wire#w1
      I_Contact( #In_Functional_Test_Even.Electrical_Current_Test_Approved_PLC_Functional_Test_30 )
      wire#w2
      S_Move(in := 'REPROVADO', out => #Functional_Tests_Panels[30].Functional_Test)
   END_RUNG
   RUNG wire#w1
      I_Contact( #In_Functional_Test_Even.Visual_Test_Approved_PLC_Functional_Test_30 )
   END_RUNG wire#w2
   // the same network as SCL:
   #_w1 := #In_Functional_Test_Even.Star_Test_PLC_Functional_Test_30 AND NOT #Aux_Trigger_30;   // rising edge of #In_Functional_Test_Even.Star_Test_PLC_Functional_Test_30
   #Aux_Trigger_30 := #In_Functional_Test_Even.Star_Test_PLC_Functional_Test_30;
   IF #_w1 THEN
       #Functional_Tests_Panels[30].Water_Fountain := #Water_Fountain;
       #Functional_Tests_Panels[30].Serial_Number := #Serial_Number;
   END_IF;
   IF #In_Functional_Test_Even.Star_Test_PLC_Functional_Test_30 THEN
       #Functional_Tests_Panels[30].Read_Electrical_Voltage := #Read_Electrial_Voltage;
   END_IF;
   IF #In_Functional_Test_Even.Star_Test_PLC_Functional_Test_30 AND NOT #In_Functional_Test_Even.Electrical_Current_Test_Approved_PLC_Functional_Test_30 THEN
       #Functional_Tests_Panels[30].Electrical_Current_Test := 'REPROVADO';
       #Functional_Tests_Panels[30].Read_Electrical_Current := #In_Functional_Test_Even.Electrical_Current_Read_PLC_Functional_Test_30;
   END_IF;
   IF #In_Functional_Test_Even.Star_Test_PLC_Functional_Test_30 AND #In_Functional_Test_Even.Electrical_Current_Test_Approved_PLC_Functional_Test_30 THEN
       #Functional_Tests_Panels[30].Electrical_Current_Test := 'APROVADO';
   END_IF;
   IF #In_Functional_Test_Even.Star_Test_PLC_Functional_Test_30 AND #In_Functional_Test_Even.Visual_Test_Approved_PLC_Functional_Test_30 THEN
       #Functional_Tests_Panels[30].Visual_Test := 'APROVADO';
   END_IF;
   IF #In_Functional_Test_Even.Star_Test_PLC_Functional_Test_30 AND NOT #In_Functional_Test_Even.Visual_Test_Approved_PLC_Functional_Test_30 THEN
       #Functional_Tests_Panels[30].Visual_Test := 'REPROVADO';
   END_IF;
   IF #In_Functional_Test_Even.Star_Test_PLC_Functional_Test_30 AND #In_Functional_Test_Even.Electrical_Current_Test_Approved_PLC_Functional_Test_30 AND #In_Functional_Test_Even.Visual_Test_Approved_PLC_Functional_Test_30 THEN
       #Functional_Tests_Panels[30].Functional_Test := 'APROVADO';
   END_IF;
   IF #In_Functional_Test_Even.Star_Test_PLC_Functional_Test_30 AND (NOT #In_Functional_Test_Even.Electrical_Current_Test_Approved_PLC_Functional_Test_30 OR NOT #In_Functional_Test_Even.Visual_Test_Approved_PLC_Functional_Test_30) THEN
       #Functional_Tests_Panels[30].Functional_Test := 'REPROVADO';
   END_IF;
END_REGION

REGION Network 31: Got married
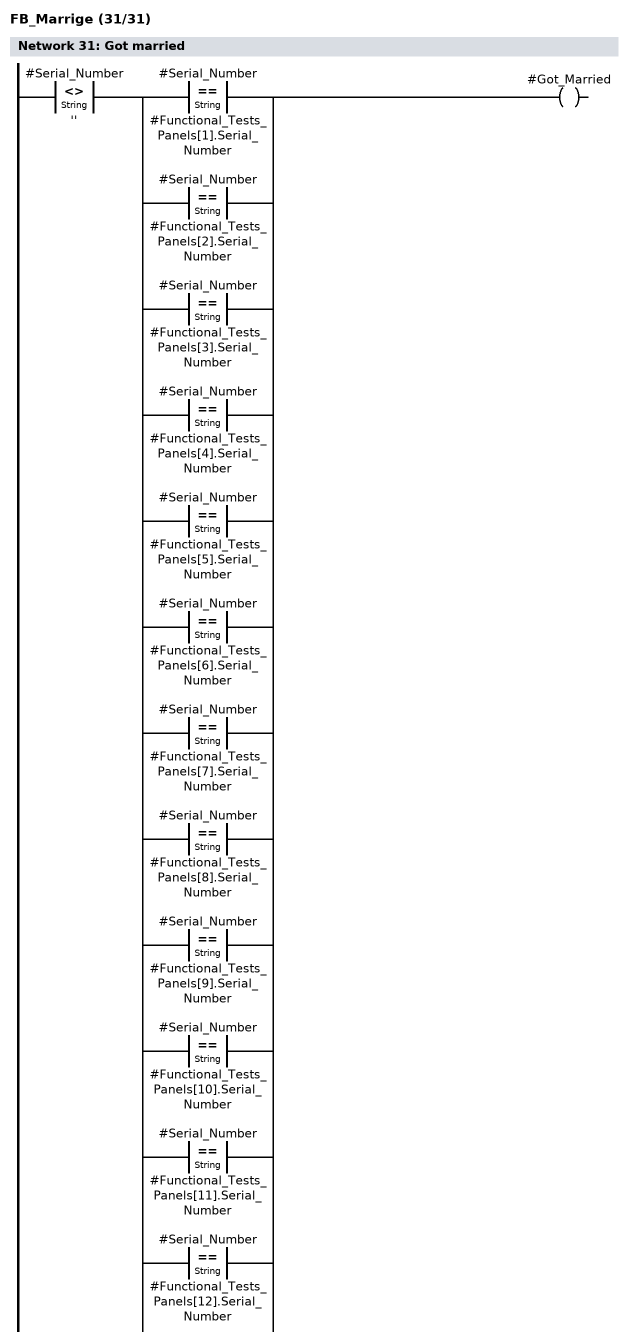
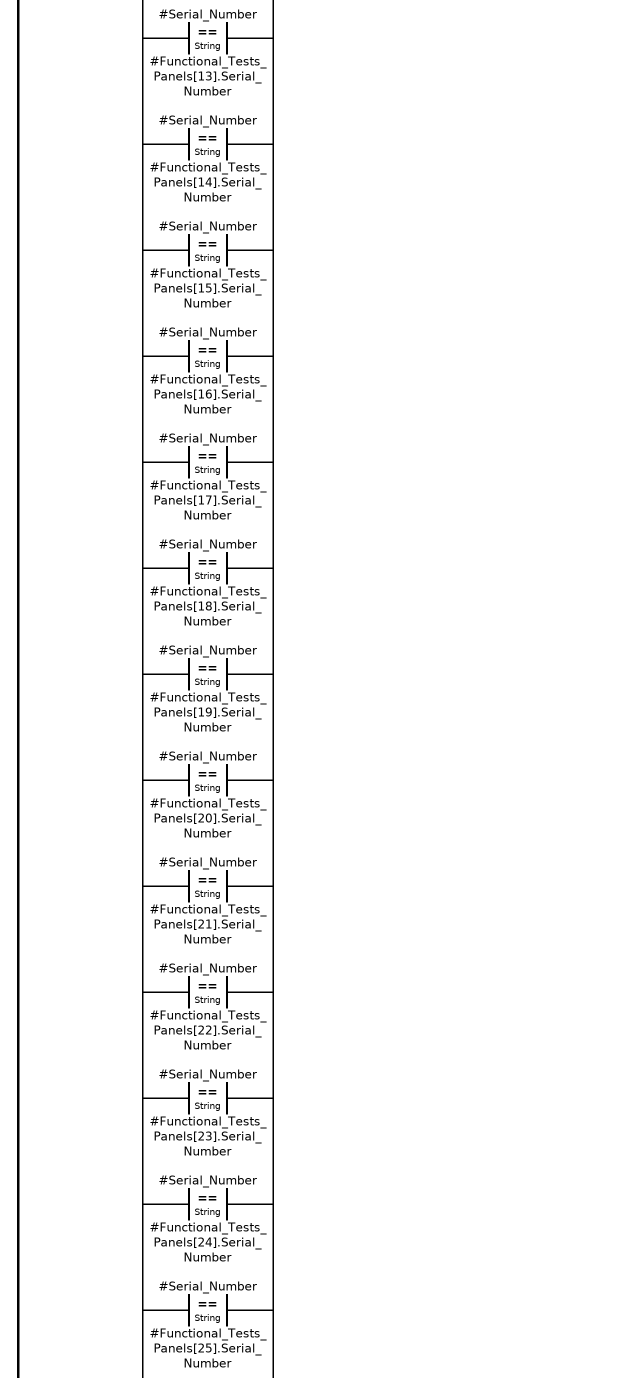
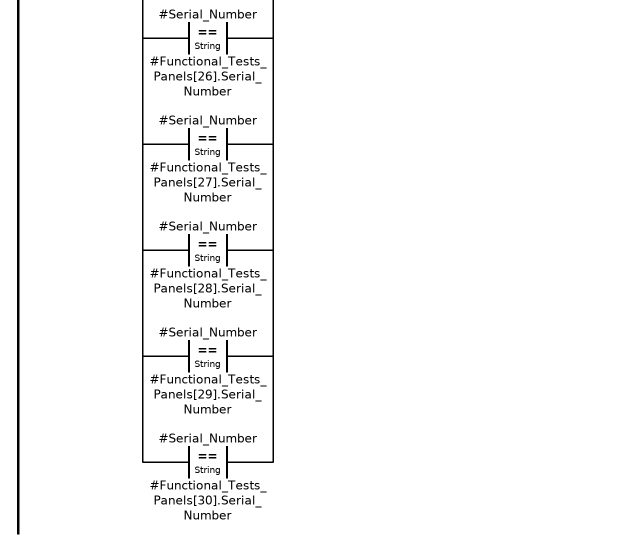
   RUNG wire#powerrail
      { S7_Templates := "SrcType := String" } NE_Contact(in1 := #Serial_Number, in2 := '')
      wire#w1
      { S7_Templates := "SrcType := String" } EQ_Contact(in1 := #Serial_Number, in2 := #Functional_Tests_Panels[1].Serial_Number)
      wire#w2
      Coil( #Got_Married )
   END_RUNG
   RUNG wire#w1
      { S7_Templates := "SrcType := String" } EQ_Contact(in1 := #Serial_Number, in2 := #Functional_Tests_Panels[2].Serial_Number)
   END_RUNG wire#w2
   RUNG wire#w1
      { S7_Templates := "SrcType := String" } EQ_Contact(in1 := #Serial_Number, in2 := #Functional_Tests_Panels[3].Serial_Number)
   END_RUNG wire#w2
   RUNG wire#w1
      { S7_Templates := "SrcType := String" } EQ_Contact(in1 := #Serial_Number, in2 := #Functional_Tests_Panels[4].Serial_Number)
   END_RUNG wire#w2
   RUNG wire#w1
      { S7_Templates := "SrcType := String" } EQ_Contact(in1 := #Serial_Number, in2 := #Functional_Tests_Panels[5].Serial_Number)
   END_RUNG wire#w2
   RUNG wire#w1
      { S7_Templates := "SrcType := String" } EQ_Contact(in1 := #Serial_Number, in2 := #Functional_Tests_Panels[6].Serial_Number)
   END_RUNG wire#w2
   RUNG wire#w1
      { S7_Templates := "SrcType := String" } EQ_Contact(in1 := #Serial_Number, in2 := #Functional_Tests_Panels[7].Serial_Number)
   END_RUNG wire#w2
   RUNG wire#w1
      { S7_Templates := "SrcType := String" } EQ_Contact(in1 := #Serial_Number, in2 := #Functional_Tests_Panels[8].Serial_Number)
   END_RUNG wire#w2
   RUNG wire#w1
      { S7_Templates := "SrcType := String" } EQ_Contact(in1 := #Serial_Number, in2 := #Functional_Tests_Panels[9].Serial_Number)
   END_RUNG wire#w2
   RUNG wire#w1
      { S7_Templates := "SrcType := String" } EQ_Contact(in1 := #Serial_Number, in2 := #Functional_Tests_Panels[10].Serial_Number)
   END_RUNG wire#w2
   RUNG wire#w1
      { S7_Templates := "SrcType := String" } EQ_Contact(in1 := #Serial_Number, in2 := #Functional_Tests_Panels[11].Serial_Number)
   END_RUNG wire#w2
   RUNG wire#w1
      { S7_Templates := "SrcType := String" } EQ_Contact(in1 := #Serial_Number, in2 := #Functional_Tests_Panels[12].Serial_Number)
   END_RUNG wire#w2
   RUNG wire#w1
      { S7_Templates := "SrcType := String" } EQ_Contact(in1 := #Serial_Number, in2 := #Functional_Tests_Panels[13].Serial_Number)
   END_RUNG wire#w2
   RUNG wire#w1
      { S7_Templates := "SrcType := String" } EQ_Contact(in1 := #Serial_Number, in2 := #Functional_Tests_Panels[14].Serial_Number)
   END_RUNG wire#w2
   RUNG wire#w1
      { S7_Templates := "SrcType := String" } EQ_Contact(in1 := #Serial_Number, in2 := #Functional_Tests_Panels[15].Serial_Number)
   END_RUNG wire#w2
   RUNG wire#w1
      { S7_Templates := "SrcType := String" } EQ_Contact(in1 := #Serial_Number, in2 := #Functional_Tests_Panels[16].Serial_Number)
   END_RUNG wire#w2
   RUNG wire#w1
      { S7_Templates := "SrcType := String" } EQ_Contact(in1 := #Serial_Number, in2 := #Functional_Tests_Panels[17].Serial_Number)
   END_RUNG wire#w2
   RUNG wire#w1
      { S7_Templates := "SrcType := String" } EQ_Contact(in1 := #Serial_Number, in2 := #Functional_Tests_Panels[18].Serial_Number)
   END_RUNG wire#w2
   RUNG wire#w1
      { S7_Templates := "SrcType := String" } EQ_Contact(in1 := #Serial_Number, in2 := #Functional_Tests_Panels[19].Serial_Number)
   END_RUNG wire#w2
   RUNG wire#w1
      { S7_Templates := "SrcType := String" } EQ_Contact(in1 := #Serial_Number, in2 := #Functional_Tests_Panels[20].Serial_Number)
   END_RUNG wire#w2
   RUNG wire#w1
      { S7_Templates := "SrcType := String" } EQ_Contact(in1 := #Serial_Number, in2 := #Functional_Tests_Panels[21].Serial_Number)
   END_RUNG wire#w2
   RUNG wire#w1
      { S7_Templates := "SrcType := String" } EQ_Contact(in1 := #Serial_Number, in2 := #Functional_Tests_Panels[22].Serial_Number)
   END_RUNG wire#w2
   RUNG wire#w1
      { S7_Templates := "SrcType := String" } EQ_Contact(in1 := #Serial_Number, in2 := #Functional_Tests_Panels[23].Serial_Number)
   END_RUNG wire#w2
   RUNG wire#w1
      { S7_Templates := "SrcType := String" } EQ_Contact(in1 := #Serial_Number, in2 := #Functional_Tests_Panels[24].Serial_Number)
   END_RUNG wire#w2
   RUNG wire#w1
      { S7_Templates := "SrcType := String" } EQ_Contact(in1 := #Serial_Number, in2 := #Functional_Tests_Panels[25].Serial_Number)
   END_RUNG wire#w2
   RUNG wire#w1
      { S7_Templates := "SrcType := String" } EQ_Contact(in1 := #Serial_Number, in2 := #Functional_Tests_Panels[26].Serial_Number)
   END_RUNG wire#w2
   RUNG wire#w1
      { S7_Templates := "SrcType := String" } EQ_Contact(in1 := #Serial_Number, in2 := #Functional_Tests_Panels[27].Serial_Number)
   END_RUNG wire#w2
   RUNG wire#w1
      { S7_Templates := "SrcType := String" } EQ_Contact(in1 := #Serial_Number, in2 := #Functional_Tests_Panels[28].Serial_Number)
   END_RUNG wire#w2
   RUNG wire#w1
      { S7_Templates := "SrcType := String" } EQ_Contact(in1 := #Serial_Number, in2 := #Functional_Tests_Panels[29].Serial_Number)
   END_RUNG wire#w2
   RUNG wire#w1
      { S7_Templates := "SrcType := String" } EQ_Contact(in1 := #Serial_Number, in2 := #Functional_Tests_Panels[30].Serial_Number)
   END_RUNG wire#w2
   // the same network as SCL:
   #Got_Married := (#Serial_Number <> '') AND ((#Serial_Number = #Functional_Tests_Panels[1].Serial_Number) OR (#Serial_Number = #Functional_Tests_Panels[2].Serial_Number) OR (#Serial_Number = #Functional_Tests_Panels[3].Serial_Number) OR (#Serial_Number = #Functional_Tests_Panels[4].Serial_Number) OR (#Serial_Number = #Functional_Tests_Panels[5].Serial_Number) OR (#Serial_Number = #Functional_Tests_Panels[6].Serial_Number) OR (#Serial_Number = #Functional_Tests_Panels[7].Serial_Number) OR (#Serial_Number = #Functional_Tests_Panels[8].Serial_Number) OR (#Serial_Number = #Functional_Tests_Panels[9].Serial_Number) OR (#Serial_Number = #Functional_Tests_Panels[10].Serial_Number) OR (#Serial_Number = #Functional_Tests_Panels[11].Serial_Number) OR (#Serial_Number = #Functional_Tests_Panels[12].Serial_Number) OR (#Serial_Number = #Functional_Tests_Panels[13].Serial_Number) OR (#Serial_Number = #Functional_Tests_Panels[14].Serial_Number) OR (#Serial_Number = #Functional_Tests_Panels[15].Serial_Number) OR (#Serial_Number = #Functional_Tests_Panels[16].Serial_Number) OR (#Serial_Number = #Functional_Tests_Panels[17].Serial_Number) OR (#Serial_Number = #Functional_Tests_Panels[18].Serial_Number) OR (#Serial_Number = #Functional_Tests_Panels[19].Serial_Number) OR (#Serial_Number = #Functional_Tests_Panels[20].Serial_Number) OR (#Serial_Number = #Functional_Tests_Panels[21].Serial_Number) OR (#Serial_Number = #Functional_Tests_Panels[22].Serial_Number) OR (#Serial_Number = #Functional_Tests_Panels[23].Serial_Number) OR (#Serial_Number = #Functional_Tests_Panels[24].Serial_Number) OR (#Serial_Number = #Functional_Tests_Panels[25].Serial_Number) OR (#Serial_Number = #Functional_Tests_Panels[26].Serial_Number) OR (#Serial_Number = #Functional_Tests_Panels[27].Serial_Number) OR (#Serial_Number = #Functional_Tests_Panels[28].Serial_Number) OR (#Serial_Number = #Functional_Tests_Panels[29].Serial_Number) OR (#Serial_Number = #Functional_Tests_Panels[30].Serial_Number));
END_REGION
END_FUNCTION_BLOCK

FUNCTION_BLOCK "FB_Search_Water_Foutain"   // FB9, LAD
{ S7_Optimized_Access := 'TRUE' }
// stored: MemoryReserve 100, SetENOAutomatically false
   VAR_INPUT
      Trigger_Read_Serial_Number_Exit_Functional_Test : Bool;
      Serial_Number : String[17];
      Functional_Tests_Panels : Array[0..31] of "Functional_Test";
   END_VAR
   VAR_OUTPUT
      Found_Functional_Test : Bool;
      Water_Foutain_Fail_Functional_Test : Bool;
      DataLog_Write : Bool;
      i : SInt;
      Search_Functional_Test : "Functional_Test";
      Reset_PLC_Functional_Test : Array[0..31] of Bool;
   END_VAR
   VAR
      Timer_Delay_Write_DataLog { S7_SetPoint := 'True'} : TON_TIME;
   END_VAR
   // Functional_Tests_Panels[0].Panel_Number := 0;
   // Functional_Tests_Panels[1].Panel_Number := 1;
   // Functional_Tests_Panels[2].Panel_Number := 2;
   // Functional_Tests_Panels[3].Panel_Number := 3;
   // Functional_Tests_Panels[4].Panel_Number := 4;
   // Functional_Tests_Panels[5].Panel_Number := 5;
   // Functional_Tests_Panels[6].Panel_Number := 6;
   // Functional_Tests_Panels[7].Panel_Number := 7;
   // Functional_Tests_Panels[8].Panel_Number := 8;
   // Functional_Tests_Panels[9].Panel_Number := 9;
   // Functional_Tests_Panels[10].Panel_Number := 10;
   // Functional_Tests_Panels[11].Panel_Number := 11;
   // Functional_Tests_Panels[12].Panel_Number := 12;
   // Functional_Tests_Panels[13].Panel_Number := 13;
   // Functional_Tests_Panels[14].Panel_Number := 14;
   // Functional_Tests_Panels[15].Panel_Number := 15;
   // Functional_Tests_Panels[16].Panel_Number := 16;
   // Functional_Tests_Panels[17].Panel_Number := 17;
   // Functional_Tests_Panels[18].Panel_Number := 18;
   // Functional_Tests_Panels[19].Panel_Number := 19;
   // Functional_Tests_Panels[20].Panel_Number := 20;
   // Functional_Tests_Panels[21].Panel_Number := 21;
   // Functional_Tests_Panels[22].Panel_Number := 22;
   // Functional_Tests_Panels[23].Panel_Number := 23;
   // Functional_Tests_Panels[24].Panel_Number := 24;
   // Functional_Tests_Panels[25].Panel_Number := 25;
   // Functional_Tests_Panels[26].Panel_Number := 26;
   // Functional_Tests_Panels[27].Panel_Number := 27;
   // Functional_Tests_Panels[28].Panel_Number := 28;
   // Functional_Tests_Panels[29].Panel_Number := 29;
   // Functional_Tests_Panels[30].Panel_Number := 30;
   // Functional_Tests_Panels[31].Panel_Number := 31;
   VAR_TEMP   // added for the SCL form of the ladder/FBD networks
      _w1 : Bool;
   END_VAR
BEGIN

REGION Network 1
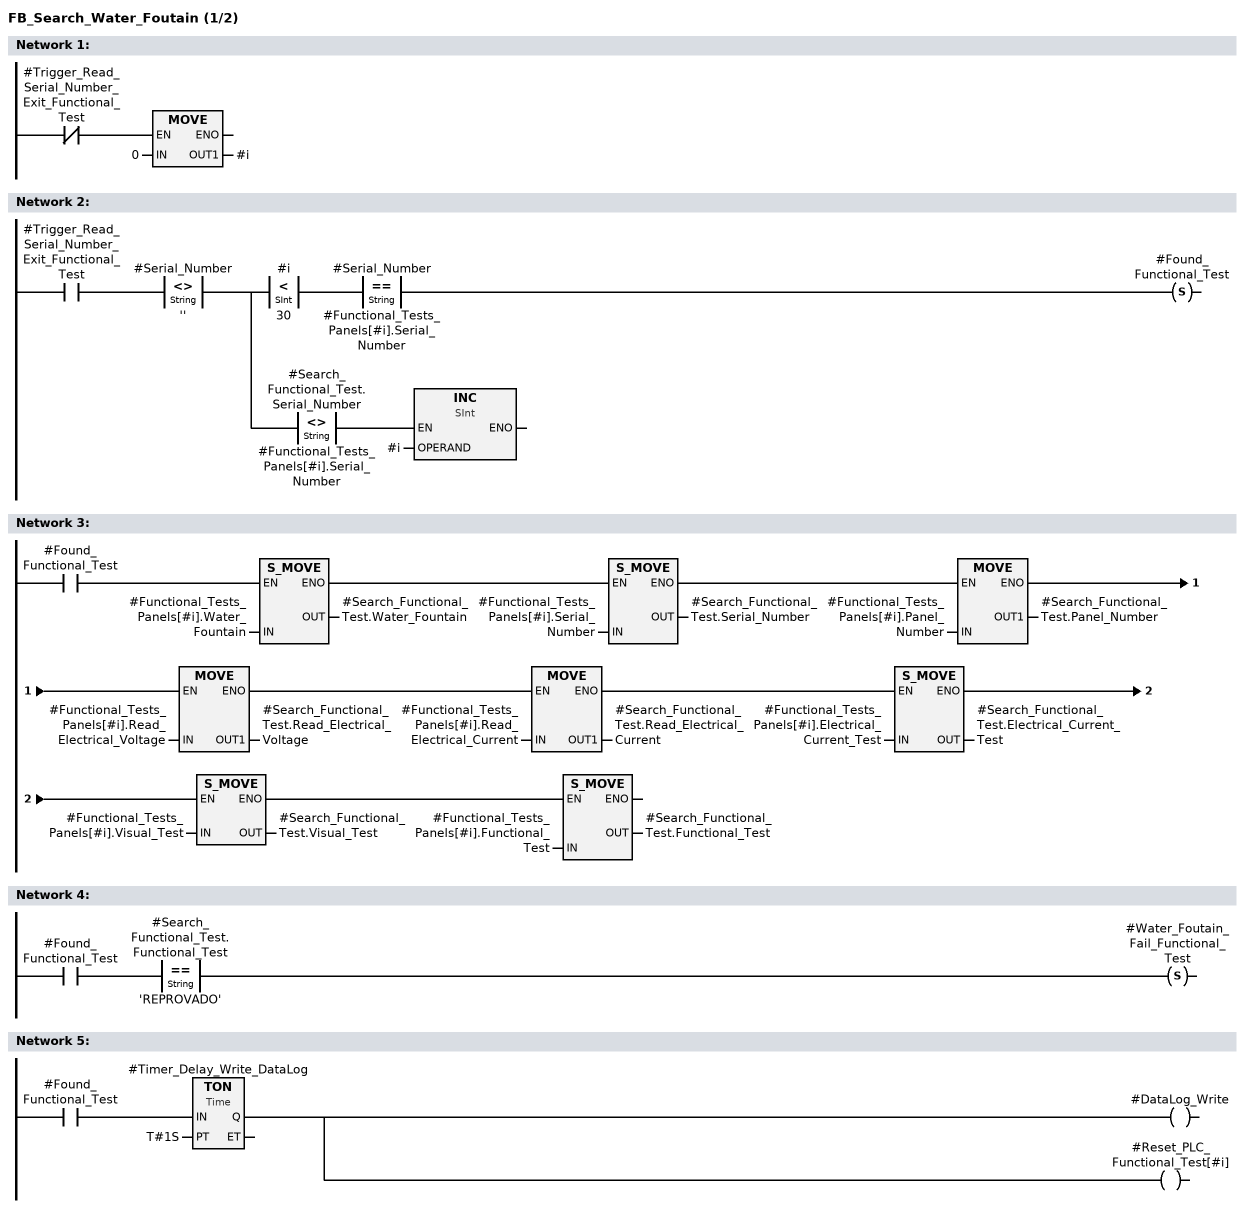
   RUNG wire#powerrail
      I_Contact( #Trigger_Read_Serial_Number_Exit_Functional_Test )
      Move(in := 0, out1 => #i)
   END_RUNG
   // the same network as SCL:
   IF NOT #Trigger_Read_Serial_Number_Exit_Functional_Test THEN #i := 0; END_IF;
END_REGION

REGION Network 2
   RUNG wire#powerrail
      Contact( #Trigger_Read_Serial_Number_Exit_Functional_Test )
      { S7_Templates := "SrcType := String" } NE_Contact(in1 := #Serial_Number, in2 := '')
      wire#w1
      { S7_Templates := "SrcType := SInt" } LT_Contact(in1 := #i, in2 := 30)
      { S7_Templates := "SrcType := String" } EQ_Contact(in1 := #Serial_Number, in2 := #Functional_Tests_Panels[#i].Serial_Number)
      S_Coil( #Found_Functional_Test )
   END_RUNG
   RUNG wire#w1
      { S7_Templates := "SrcType := String" } NE_Contact(in1 := #Search_Functional_Test.Serial_Number, in2 := #Functional_Tests_Panels[#i].Serial_Number)
      { S7_Templates := "DestType := SInt" } Inc( #i )
   END_RUNG
   // the same network as SCL:
   #_w1 := #Trigger_Read_Serial_Number_Exit_Functional_Test AND (#Serial_Number <> '');
   IF #_w1 AND (#i < 30) AND (#Serial_Number = #Functional_Tests_Panels[#i].Serial_Number) THEN
       #Found_Functional_Test := TRUE;
   END_IF;
   IF #_w1 AND (#Search_Functional_Test.Serial_Number <> #Functional_Tests_Panels[#i].Serial_Number) THEN
       #i := #i + 1;
   END_IF;
END_REGION

REGION Network 3
   RUNG wire#powerrail
      Contact( #Found_Functional_Test )
      S_Move(in := #Functional_Tests_Panels[#i].Water_Fountain, out => #Search_Functional_Test.Water_Fountain)
      S_Move(in := #Functional_Tests_Panels[#i].Serial_Number, out => #Search_Functional_Test.Serial_Number)
      Move(in := #Functional_Tests_Panels[#i].Panel_Number, out1 => #Search_Functional_Test.Panel_Number)
      Move(in := #Functional_Tests_Panels[#i].Read_Electrical_Voltage, out1 => #Search_Functional_Test.Read_Electrical_Voltage)
      Move(in := #Functional_Tests_Panels[#i].Read_Electrical_Current, out1 => #Search_Functional_Test.Read_Electrical_Current)
      S_Move(in := #Functional_Tests_Panels[#i].Electrical_Current_Test, out => #Search_Functional_Test.Electrical_Current_Test)
      S_Move(in := #Functional_Tests_Panels[#i].Visual_Test, out => #Search_Functional_Test.Visual_Test)
      S_Move(in := #Functional_Tests_Panels[#i].Functional_Test, out => #Search_Functional_Test.Functional_Test)
   END_RUNG
   // the same network as SCL:
   IF #Found_Functional_Test THEN
       #Search_Functional_Test.Water_Fountain := #Functional_Tests_Panels[#i].Water_Fountain;
       #Search_Functional_Test.Serial_Number := #Functional_Tests_Panels[#i].Serial_Number;
       #Search_Functional_Test.Panel_Number := #Functional_Tests_Panels[#i].Panel_Number;
       #Search_Functional_Test.Read_Electrical_Voltage := #Functional_Tests_Panels[#i].Read_Electrical_Voltage;
       #Search_Functional_Test.Read_Electrical_Current := #Functional_Tests_Panels[#i].Read_Electrical_Current;
       #Search_Functional_Test.Electrical_Current_Test := #Functional_Tests_Panels[#i].Electrical_Current_Test;
       #Search_Functional_Test.Visual_Test := #Functional_Tests_Panels[#i].Visual_Test;
       #Search_Functional_Test.Functional_Test := #Functional_Tests_Panels[#i].Functional_Test;
   END_IF;
END_REGION

REGION Network 4
   RUNG wire#powerrail
      Contact( #Found_Functional_Test )
      { S7_Templates := "SrcType := String" } EQ_Contact(in1 := #Search_Functional_Test.Functional_Test, in2 := 'REPROVADO')
      S_Coil( #Water_Foutain_Fail_Functional_Test )
   END_RUNG
   // the same network as SCL:
   IF #Found_Functional_Test AND (#Search_Functional_Test.Functional_Test = 'REPROVADO') THEN
       #Water_Foutain_Fail_Functional_Test := TRUE;
   END_IF;
END_REGION

REGION Network 5
   RUNG wire#powerrail
      Contact( #Found_Functional_Test )
      { S7_Templates := "time_type := Time" } #Timer_Delay_Write_DataLog.TON(pt := T#1S, et =>)
      wire#w1
      Coil( #DataLog_Write )
   END_RUNG
   RUNG wire#w1
      Coil( #Reset_PLC_Functional_Test[#i] )
   END_RUNG
   // the same network as SCL:
   #Timer_Delay_Write_DataLog(IN := #Found_Functional_Test, PT := T#1S);   // TON
   #DataLog_Write := #Timer_Delay_Write_DataLog.Q;
   #Reset_PLC_Functional_Test[#i] := #Timer_Delay_Write_DataLog.Q;
END_REGION

REGION Network 6
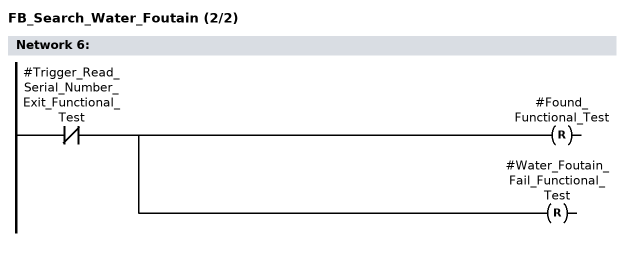
   RUNG wire#powerrail
      I_Contact( #Trigger_Read_Serial_Number_Exit_Functional_Test )
      wire#w1
      R_Coil( #Found_Functional_Test )
   END_RUNG
   RUNG wire#w1
      R_Coil( #Water_Foutain_Fail_Functional_Test )
   END_RUNG
   // the same network as SCL:
   IF NOT #Trigger_Read_Serial_Number_Exit_Functional_Test THEN
       #Found_Functional_Test := FALSE;
       #Water_Foutain_Fail_Functional_Test := FALSE;
   END_IF;
END_REGION
END_FUNCTION_BLOCK

FUNCTION_BLOCK "FB_DataLog"   // FB10, LAD
{ S7_Optimized_Access := 'TRUE' }
// stored: AutoNumber false, MemoryReserve 100, SetENOAutomatically false
   VAR_INPUT
      DataLogCreate_REQ : Bool;
      DataLogOpen_REQ : Bool;
      DataLogWrite_REQ : Bool;
      DataLogClose_REQ : Bool;
      DataLogClear_REQ : Bool;
      DataLogDelete_REQ : Bool;
   END_VAR
   VAR_OUTPUT
      DataLogCreate_DONE : Bool;
      DataLogCreate_BUSY : Bool;
      DataLogCreate_ERROR : Bool;
      DataLogCreate_STATUS : Word;
      DataLogOpen_DONE : Bool;
      DataLogOpen_BUSY : Bool;
      DataLogOpen_ERROR : Bool;
      DataLogOpen_STATUS : Word;
      DataLogWrite_DONE : Bool;
      DataLogWrite_BUSY : Bool;
      DataLogWrite_ERROR : Bool;
      DataLogWrite_STATUS : Word;
      DataLogClose_DONE : Bool;
      DataLogClose_BUSY : Bool;
      DataLogClose_ERROR : Bool;
      DataLogClose_STATUS : Word;
      DataLogClear_DONE : Bool;
      DataLogClear_BUSY : Bool;
      DataLogClear_ERROR : Bool;
      DataLogClear_STATUS : Word;
      DataLogDelete_DONE : Bool;
      DataLogDelete_BUSY : Bool;
      DataLogDelete_ERROR : Bool;
      DataLogDelete_STATUS : Word;
   END_VAR
   VAR_IN_OUT
      ID : DWord;
      "NAME" : Variant;
      DataLogCreate_HEADER : Variant;
      DATA : Variant;
   END_VAR
   VAR
      Enable_DataLogOpen : Bool;
      Enable_DataLogWrite : Bool;
      Axiliar_P_Trig_0 : Bool;
      Axiliar_P_Trig_1 : Bool;
      Axiliar_P_Trig_2 : Bool;
      Axiliar_P_Trig_3 : Bool;
      Axiliar_P_Trig_4 : Bool;
      Axiliar_P_Trig_5 : Bool;
      Axiliar_P_Trig_6 : Bool;
      Axiliar_P_Trig_7 : Bool;
      Axiliar_P_Trig_8 : Bool;
      DataLogCreate_Instance { S7_SetPoint := 'True'} : DataLogCreate;
      DataLogOpen_Instance { S7_SetPoint := 'True'} : DataLogOpen;
      DataLogWrite_Instance { S7_SetPoint := 'True'} : DataLogWrite;
      DataLogClose_Instance { S7_SetPoint := 'True'} : DataLogClose;
      DataLogClear_Instance { S7_SetPoint := 'True'} : DataLogClear;
      DataLogDelete_Instance { S7_SetPoint := 'True'} : DataLogDelete;
   END_VAR
   VAR_TEMP   // added for the SCL form of the ladder/FBD networks
      _w1 : Bool;
      _w2 : Bool;
      _w3 : Bool;
   END_VAR
BEGIN

REGION Network 1: Create DataLog
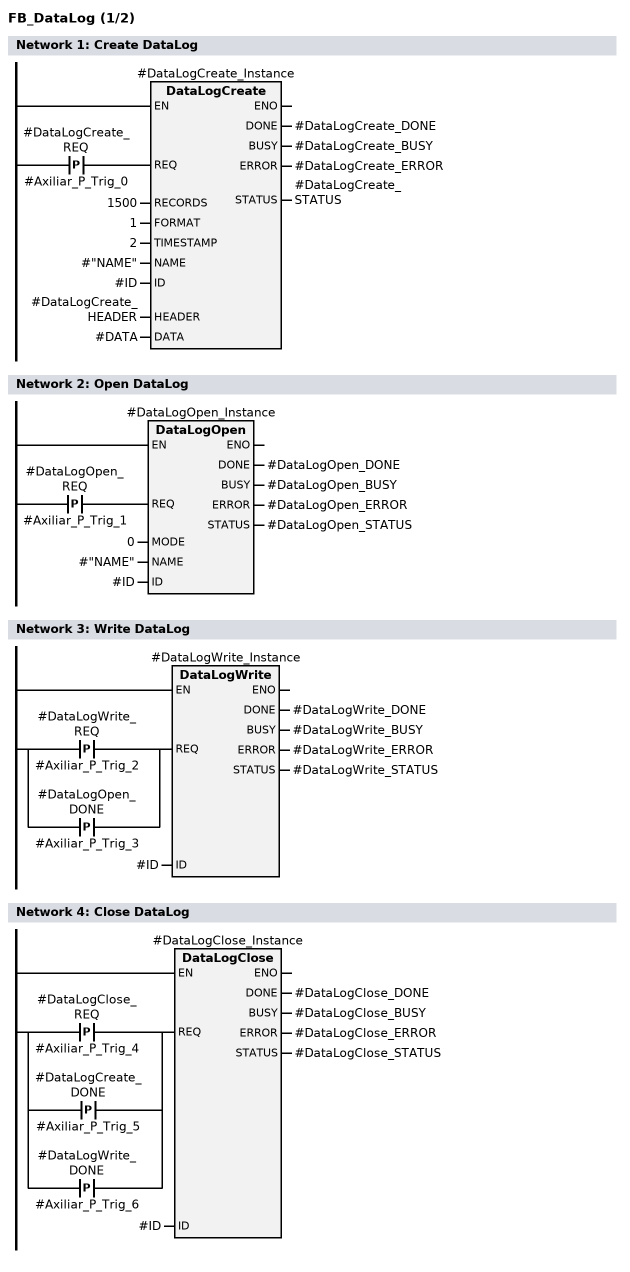
   RUNG wire#powerrail
      #DataLogCreate_Instance.DataLogCreate(REQ := wire#w1, RECORDS := 1500, FORMAT := 1, TIMESTAMP := 2, "NAME" := #"NAME", ID := #ID, HEADER := #DataLogCreate_HEADER, DATA := #DATA, DONE => #DataLogCreate_DONE, BUSY => #DataLogCreate_BUSY, ERROR => #DataLogCreate_ERROR, STATUS => #DataLogCreate_STATUS)
   END_RUNG
   RUNG wire#powerrail
      P_Contact(operand := #DataLogCreate_REQ, bit := #Axiliar_P_Trig_0)
   END_RUNG wire#w1
   // the same network as SCL:
   #_w1 := #DataLogCreate_REQ AND NOT #Axiliar_P_Trig_0;   // rising edge of #DataLogCreate_REQ
   #Axiliar_P_Trig_0 := #DataLogCreate_REQ;
   #DataLogCreate_Instance(REQ := #_w1,   // DataLogCreate
                           RECORDS := 1500,
                           FORMAT := 1,
                           TIMESTAMP := 2,
                           "NAME" := #"NAME",
                           ID := #ID,
                           HEADER := #DataLogCreate_HEADER,
                           DATA := #DATA,
                           DONE => #DataLogCreate_DONE,
                           BUSY => #DataLogCreate_BUSY,
                           ERROR => #DataLogCreate_ERROR,
                           STATUS => #DataLogCreate_STATUS);
END_REGION

REGION Network 2: Open DataLog
   RUNG wire#powerrail
      { S7_Templates := "card := 0" } #DataLogOpen_Instance.DataLogOpen(REQ := wire#w1, MODE := 0, "NAME" := #"NAME", ID := #ID, DONE => #DataLogOpen_DONE, BUSY => #DataLogOpen_BUSY, ERROR => #DataLogOpen_ERROR, STATUS => #DataLogOpen_STATUS)
   END_RUNG
   RUNG wire#powerrail
      P_Contact(operand := #DataLogOpen_REQ, bit := #Axiliar_P_Trig_1)
   END_RUNG wire#w1
   // the same network as SCL:
   #_w1 := #DataLogOpen_REQ AND NOT #Axiliar_P_Trig_1;   // rising edge of #DataLogOpen_REQ
   #Axiliar_P_Trig_1 := #DataLogOpen_REQ;
   #DataLogOpen_Instance(REQ := #_w1,   // DataLogOpen
                         MODE := 0,
                         "NAME" := #"NAME",
                         ID := #ID,
                         DONE => #DataLogOpen_DONE,
                         BUSY => #DataLogOpen_BUSY,
                         ERROR => #DataLogOpen_ERROR,
                         STATUS => #DataLogOpen_STATUS);
END_REGION

REGION Network 3: Write DataLog
   RUNG wire#powerrail
      #DataLogWrite_Instance.DataLogWrite(REQ := wire#w1, ID := #ID, DONE => #DataLogWrite_DONE, BUSY => #DataLogWrite_BUSY, ERROR => #DataLogWrite_ERROR, STATUS => #DataLogWrite_STATUS)
   END_RUNG
   RUNG wire#powerrail
      P_Contact(operand := #DataLogWrite_REQ, bit := #Axiliar_P_Trig_2)
   END_RUNG wire#w1
   RUNG wire#powerrail
      P_Contact(operand := #DataLogOpen_DONE, bit := #Axiliar_P_Trig_3)
   END_RUNG wire#w1
   // the same network as SCL:
   #_w1 := #DataLogWrite_REQ AND NOT #Axiliar_P_Trig_2;   // rising edge of #DataLogWrite_REQ
   #Axiliar_P_Trig_2 := #DataLogWrite_REQ;
   #_w2 := #DataLogOpen_DONE AND NOT #Axiliar_P_Trig_3;   // rising edge of #DataLogOpen_DONE
   #Axiliar_P_Trig_3 := #DataLogOpen_DONE;
   #DataLogWrite_Instance(REQ := #_w1 OR #_w2,   // DataLogWrite
                          ID := #ID,
                          DONE => #DataLogWrite_DONE,
                          BUSY => #DataLogWrite_BUSY,
                          ERROR => #DataLogWrite_ERROR,
                          STATUS => #DataLogWrite_STATUS);
END_REGION

REGION Network 4: Close DataLog
   RUNG wire#powerrail
      #DataLogClose_Instance.DataLogClose(REQ := wire#w1, ID := #ID, DONE => #DataLogClose_DONE, BUSY => #DataLogClose_BUSY, ERROR => #DataLogClose_ERROR, STATUS => #DataLogClose_STATUS)
   END_RUNG
   RUNG wire#powerrail
      P_Contact(operand := #DataLogClose_REQ, bit := #Axiliar_P_Trig_4)
   END_RUNG wire#w1
   RUNG wire#powerrail
      P_Contact(operand := #DataLogCreate_DONE, bit := #Axiliar_P_Trig_5)
   END_RUNG wire#w1
   RUNG wire#powerrail
      P_Contact(operand := #DataLogWrite_DONE, bit := #Axiliar_P_Trig_6)
   END_RUNG wire#w1
   // the same network as SCL:
   #_w1 := #DataLogClose_REQ AND NOT #Axiliar_P_Trig_4;   // rising edge of #DataLogClose_REQ
   #Axiliar_P_Trig_4 := #DataLogClose_REQ;
   #_w2 := #DataLogCreate_DONE AND NOT #Axiliar_P_Trig_5;   // rising edge of #DataLogCreate_DONE
   #Axiliar_P_Trig_5 := #DataLogCreate_DONE;
   #_w3 := #DataLogWrite_DONE AND NOT #Axiliar_P_Trig_6;   // rising edge of #DataLogWrite_DONE
   #Axiliar_P_Trig_6 := #DataLogWrite_DONE;
   #DataLogClose_Instance(REQ := #_w1 OR #_w2 OR #_w3,   // DataLogClose
                          ID := #ID,
                          DONE => #DataLogClose_DONE,
                          BUSY => #DataLogClose_BUSY,
                          ERROR => #DataLogClose_ERROR,
                          STATUS => #DataLogClose_STATUS);
END_REGION

REGION Network 5: Clear DataLog
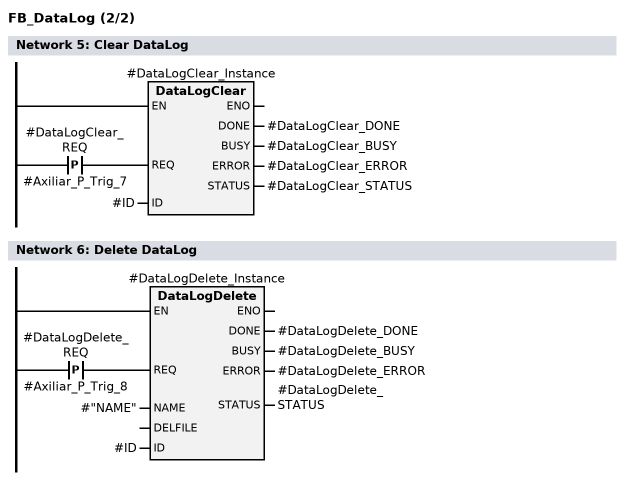
   RUNG wire#powerrail
      #DataLogClear_Instance.DataLogClear(REQ := wire#w1, ID := #ID, DONE => #DataLogClear_DONE, BUSY => #DataLogClear_BUSY, ERROR => #DataLogClear_ERROR, STATUS => #DataLogClear_STATUS)
   END_RUNG
   RUNG wire#powerrail
      P_Contact(operand := #DataLogClear_REQ, bit := #Axiliar_P_Trig_7)
   END_RUNG wire#w1
   // the same network as SCL:
   #_w1 := #DataLogClear_REQ AND NOT #Axiliar_P_Trig_7;   // rising edge of #DataLogClear_REQ
   #Axiliar_P_Trig_7 := #DataLogClear_REQ;
   #DataLogClear_Instance(REQ := #_w1,   // DataLogClear
                          ID := #ID,
                          DONE => #DataLogClear_DONE,
                          BUSY => #DataLogClear_BUSY,
                          ERROR => #DataLogClear_ERROR,
                          STATUS => #DataLogClear_STATUS);
END_REGION

REGION Network 6: Delete DataLog
   RUNG wire#powerrail
      #DataLogDelete_Instance.DataLogDelete(REQ := wire#w1, "NAME" := #"NAME", DelFile :=, ID := #ID, DONE => #DataLogDelete_DONE, BUSY => #DataLogDelete_BUSY, ERROR => #DataLogDelete_ERROR, STATUS => #DataLogDelete_STATUS)
   END_RUNG
   RUNG wire#powerrail
      P_Contact(operand := #DataLogDelete_REQ, bit := #Axiliar_P_Trig_8)
   END_RUNG wire#w1
   // the same network as SCL:
   #_w1 := #DataLogDelete_REQ AND NOT #Axiliar_P_Trig_8;   // rising edge of #DataLogDelete_REQ
   #Axiliar_P_Trig_8 := #DataLogDelete_REQ;
   #DataLogDelete_Instance(REQ := #_w1,   // DataLogDelete
                           "NAME" := #"NAME",
                           ID := #ID,
                           DONE => #DataLogDelete_DONE,
                           BUSY => #DataLogDelete_BUSY,
                           ERROR => #DataLogDelete_ERROR,
                           STATUS => #DataLogDelete_STATUS);
END_REGION
END_FUNCTION_BLOCK

FUNCTION_BLOCK "FB_HMI"   // FB11, LAD
{ S7_Optimized_Access := 'TRUE' }
// stored: AutoNumber false, MemoryReserve 100, SetENOAutomatically false
   VAR_INPUT
      Control_Screen_HMI : Word;
      Employee_Rework : String[6];
      Admin_1 : String[6] := '';
      Admin_2 : String[6];
      Admin_3 : String[6];
      Admin_4 : String[6];
      Admin_5 : String[6];
      Alarm_0 : Word;
      Alarm_1 : Word;
      Alarm_2 : Word;
   END_VAR
   VAR_OUTPUT
      Alarm : Bool;
      Job_Mailbox : Array[0..3] of Word;
   END_VAR
   VAR
      Aux_Trigger_0 : Bool;
      Aux_Trigger_1 : Bool;
      Aux_Trigger_2 : Bool;
      Aux_Trigger_3 : Bool;
      Aux_Trigger_4 : Bool;
      Aux_Trigger_5 : Bool;
      Aux_Trigger_6 : Bool;
      Aux_Trigger_7 : Bool;
      Aux_Trigger_8 : Bool;
      Aux_Trigger_9 : Bool;
      Aux_Trigger_10 : Bool;
      Everybody_Can_Access : Bool;
      Only_Admin_Can_Access : Bool;
      Control_Screen : Word;
      Timer_Delay_Change_Screen { S7_SetPoint := 'True'} : TON_TIME;
      Timer_Delay_Change_Job_Mailbox { S7_SetPoint := 'True'} : TON_TIME;
   END_VAR
   VAR CONSTANT
      Screen_1 : Word := 16#1;
      Screen_2 : Word := 16#2;
      Screen_3 : Word := 16#3;
      Screen_4 : Word := 16#4;
      Screen_5 : Word := 16#5;
      Screen_6 : Word := 16#6;
      Screen_7 : Word := 16#7;
      Screen_8 : Word := 16#8;
      Screen_9 : Word := 16#9;
      Screen_10 : Word := 16#20;
      Screen_11 : Word := 16#21;
      Screen_12 : Word := 16#22;
      Screen_13 : Word := 16#23;
      Screen_14 : Word := 16#24;
      Lau : String := 'Lau$R$00$00';
   END_VAR
   // Job_Mailbox[0] := 51;
   // Job_Mailbox[2..3] := 0;
   VAR_TEMP   // added for the SCL form of the ladder/FBD networks
      _w1 : Bool;
      _w2 : Bool;
      _w3 : Bool;
   END_VAR
BEGIN

REGION Network 1: Admin
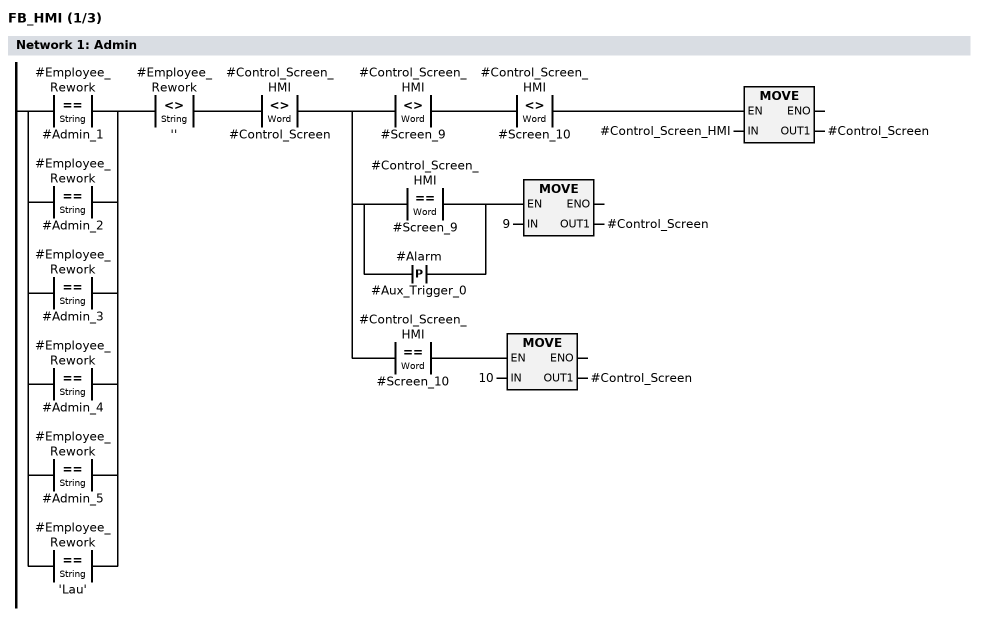
   RUNG wire#powerrail
      { S7_Templates := "SrcType := String" } EQ_Contact(in1 := #Employee_Rework, in2 := #Admin_1)
      wire#w1
      { S7_Templates := "SrcType := String" } NE_Contact(in1 := #Employee_Rework, in2 := '')
      { S7_Templates := "SrcType := Word" } NE_Contact(in1 := #Control_Screen_HMI, in2 := #Control_Screen)
      wire#w2
      { S7_Templates := "SrcType := Word" } NE_Contact(in1 := #Control_Screen_HMI, in2 := #Screen_9)
      { S7_Templates := "SrcType := Word" } NE_Contact(in1 := #Control_Screen_HMI, in2 := #Screen_10)
      Move(in := #Control_Screen_HMI, out1 => #Control_Screen)
   END_RUNG
   RUNG wire#powerrail
      { S7_Templates := "SrcType := String" } EQ_Contact(in1 := #Employee_Rework, in2 := #Admin_2)
   END_RUNG wire#w1
   RUNG wire#powerrail
      { S7_Templates := "SrcType := String" } EQ_Contact(in1 := #Employee_Rework, in2 := #Admin_3)
   END_RUNG wire#w1
   RUNG wire#powerrail
      { S7_Templates := "SrcType := String" } EQ_Contact(in1 := #Employee_Rework, in2 := #Admin_4)
   END_RUNG wire#w1
   RUNG wire#powerrail
      { S7_Templates := "SrcType := String" } EQ_Contact(in1 := #Employee_Rework, in2 := #Admin_5)
   END_RUNG wire#w1
   RUNG wire#powerrail
      { S7_Templates := "SrcType := String" } EQ_Contact(in1 := #Employee_Rework, in2 := 'Lau')
   END_RUNG wire#w1
   RUNG wire#w2
      { S7_Templates := "SrcType := Word" } EQ_Contact(in1 := #Control_Screen_HMI, in2 := #Screen_9)
      wire#w3
      Move(in := 9, out1 => #Control_Screen)
   END_RUNG
   RUNG wire#w2
      P_Contact(operand := #Alarm, bit := #Aux_Trigger_0)
   END_RUNG wire#w3
   RUNG wire#w2
      { S7_Templates := "SrcType := Word" } EQ_Contact(in1 := #Control_Screen_HMI, in2 := #Screen_10)
      Move(in := 10, out1 => #Control_Screen)
   END_RUNG
   // the same network as SCL:
   #_w1 := ((#Employee_Rework = #Admin_1) OR (#Employee_Rework = #Admin_2) OR (#Employee_Rework = #Admin_3) OR (#Employee_Rework = #Admin_4) OR (#Employee_Rework = #Admin_5) OR (#Employee_Rework = 'Lau')) AND (#Employee_Rework <> '') AND (#Control_Screen_HMI <> #Control_Screen);
   IF #_w1 AND (#Control_Screen_HMI <> #Screen_9) AND (#Control_Screen_HMI <> #Screen_10) THEN
       #Control_Screen := #Control_Screen_HMI;
   END_IF;
   #_w2 := #_w1 AND #Alarm AND NOT #Aux_Trigger_0;   // rising edge of #Alarm
   #Aux_Trigger_0 := #Alarm;
   IF (#_w1 AND (#Control_Screen_HMI = #Screen_9)) OR #_w2 THEN #Control_Screen := 9; END_IF;
   IF #_w1 AND (#Control_Screen_HMI = #Screen_10) THEN #Control_Screen := 10; END_IF;
END_REGION

REGION Network 2
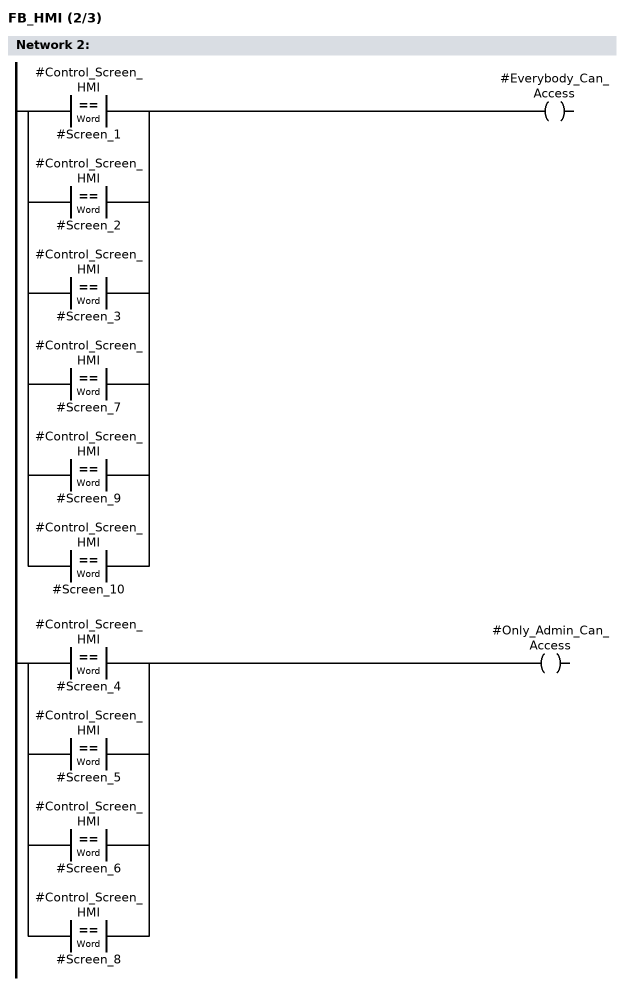
   RUNG wire#powerrail
      { S7_Templates := "SrcType := Word" } EQ_Contact(in1 := #Control_Screen_HMI, in2 := #Screen_1)
      wire#w1
      Coil( #Everybody_Can_Access )
   END_RUNG
   RUNG wire#powerrail
      { S7_Templates := "SrcType := Word" } EQ_Contact(in1 := #Control_Screen_HMI, in2 := #Screen_2)
   END_RUNG wire#w1
   RUNG wire#powerrail
      { S7_Templates := "SrcType := Word" } EQ_Contact(in1 := #Control_Screen_HMI, in2 := #Screen_3)
   END_RUNG wire#w1
   RUNG wire#powerrail
      { S7_Templates := "SrcType := Word" } EQ_Contact(in1 := #Control_Screen_HMI, in2 := #Screen_7)
   END_RUNG wire#w1
   RUNG wire#powerrail
      { S7_Templates := "SrcType := Word" } EQ_Contact(in1 := #Control_Screen_HMI, in2 := #Screen_9)
   END_RUNG wire#w1
   RUNG wire#powerrail
      { S7_Templates := "SrcType := Word" } EQ_Contact(in1 := #Control_Screen_HMI, in2 := #Screen_10)
   END_RUNG wire#w1
   RUNG wire#powerrail
      { S7_Templates := "SrcType := Word" } EQ_Contact(in1 := #Control_Screen_HMI, in2 := #Screen_4)
      wire#w2
      Coil( #Only_Admin_Can_Access )
   END_RUNG
   RUNG wire#powerrail
      { S7_Templates := "SrcType := Word" } EQ_Contact(in1 := #Control_Screen_HMI, in2 := #Screen_5)
   END_RUNG wire#w2
   RUNG wire#powerrail
      { S7_Templates := "SrcType := Word" } EQ_Contact(in1 := #Control_Screen_HMI, in2 := #Screen_6)
   END_RUNG wire#w2
   RUNG wire#powerrail
      { S7_Templates := "SrcType := Word" } EQ_Contact(in1 := #Control_Screen_HMI, in2 := #Screen_8)
   END_RUNG wire#w2
   // the same network as SCL:
   #Everybody_Can_Access := (#Control_Screen_HMI = #Screen_1) OR (#Control_Screen_HMI = #Screen_2) OR (#Control_Screen_HMI = #Screen_3) OR (#Control_Screen_HMI = #Screen_7) OR (#Control_Screen_HMI = #Screen_9) OR (#Control_Screen_HMI = #Screen_10);
   #Only_Admin_Can_Access := (#Control_Screen_HMI = #Screen_4) OR (#Control_Screen_HMI = #Screen_5) OR (#Control_Screen_HMI = #Screen_6) OR (#Control_Screen_HMI = #Screen_8);
END_REGION

REGION Network 3: Not Admin
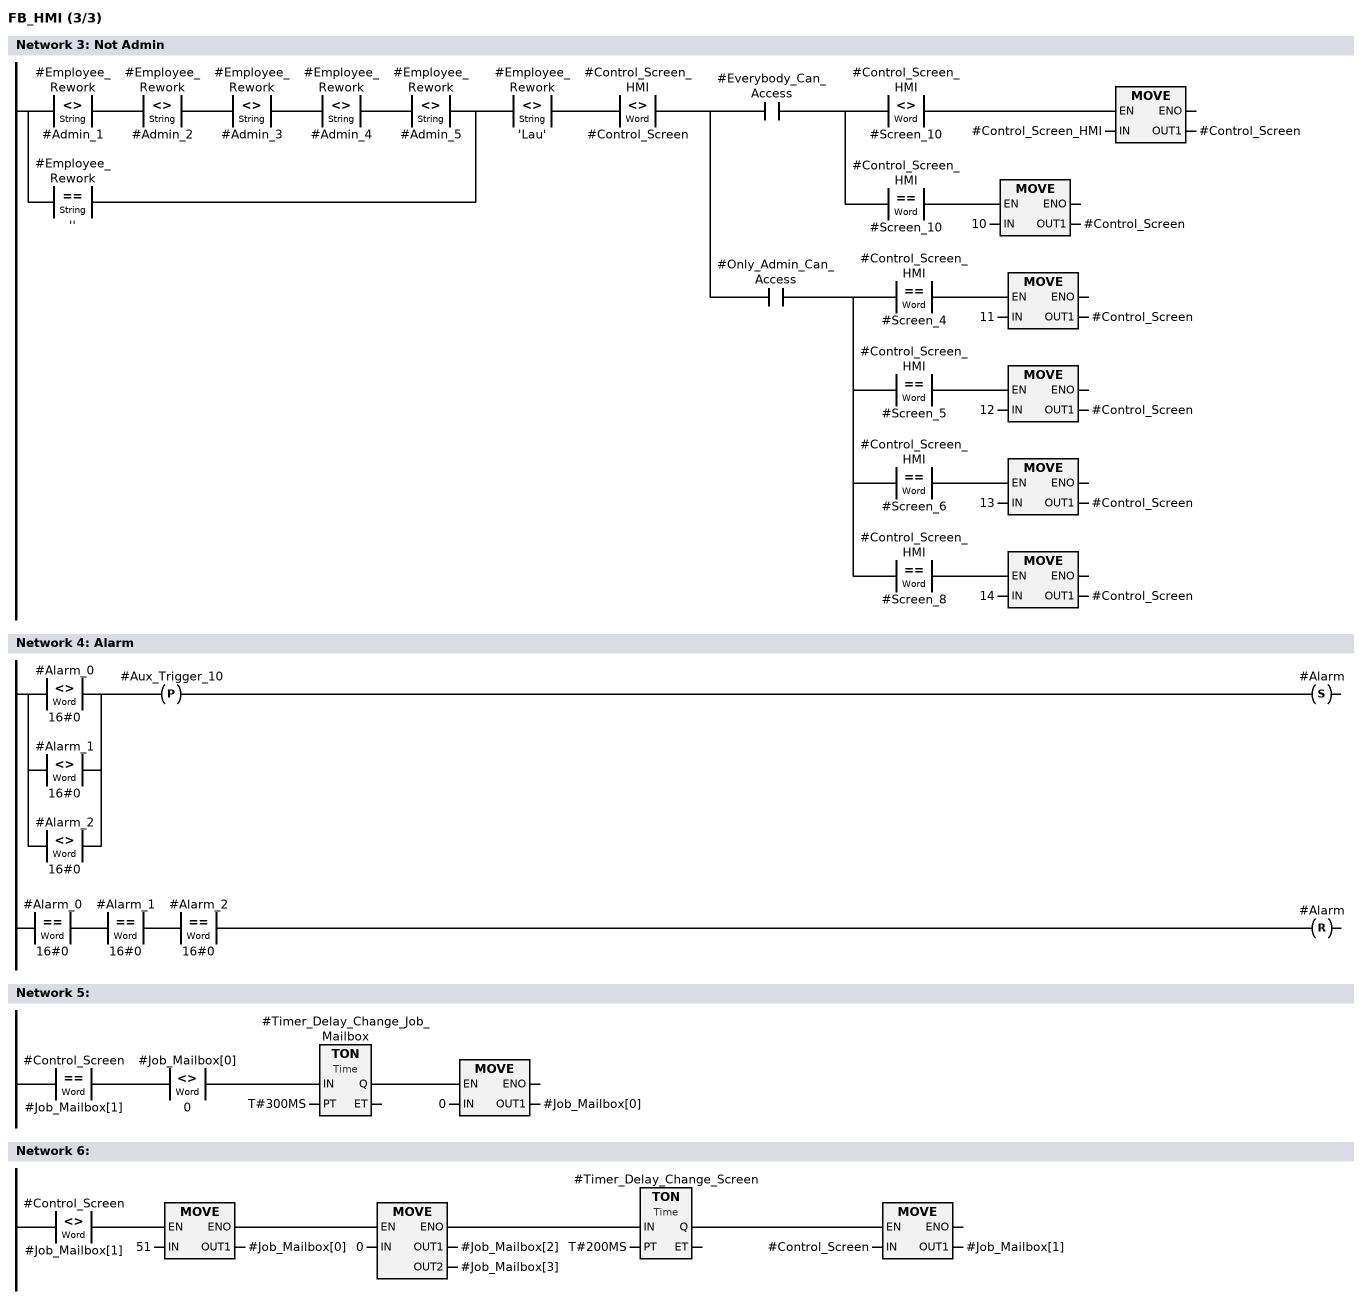
   RUNG wire#powerrail
      { S7_Templates := "SrcType := String" } NE_Contact(in1 := #Employee_Rework, in2 := #Admin_1)
      { S7_Templates := "SrcType := String" } NE_Contact(in1 := #Employee_Rework, in2 := #Admin_2)
      { S7_Templates := "SrcType := String" } NE_Contact(in1 := #Employee_Rework, in2 := #Admin_3)
      { S7_Templates := "SrcType := String" } NE_Contact(in1 := #Employee_Rework, in2 := #Admin_4)
      { S7_Templates := "SrcType := String" } NE_Contact(in1 := #Employee_Rework, in2 := #Admin_5)
      wire#w1
      { S7_Templates := "SrcType := String" } NE_Contact(in1 := #Employee_Rework, in2 := 'Lau')
      { S7_Templates := "SrcType := Word" } NE_Contact(in1 := #Control_Screen_HMI, in2 := #Control_Screen)
      wire#w2
      Contact( #Everybody_Can_Access )
      wire#w3
      { S7_Templates := "SrcType := Word" } NE_Contact(in1 := #Control_Screen_HMI, in2 := #Screen_10)
      Move(in := #Control_Screen_HMI, out1 => #Control_Screen)
   END_RUNG
   RUNG wire#powerrail
      { S7_Templates := "SrcType := String" } EQ_Contact(in1 := #Employee_Rework, in2 := '')
   END_RUNG wire#w1
   RUNG wire#w3
      { S7_Templates := "SrcType := Word" } EQ_Contact(in1 := #Control_Screen_HMI, in2 := #Screen_10)
      Move(in := 10, out1 => #Control_Screen)
   END_RUNG
   RUNG wire#w2
      Contact( #Only_Admin_Can_Access )
      wire#w4
      { S7_Templates := "SrcType := Word" } EQ_Contact(in1 := #Control_Screen_HMI, in2 := #Screen_4)
      Move(in := 11, out1 => #Control_Screen)
   END_RUNG
   RUNG wire#w4
      { S7_Templates := "SrcType := Word" } EQ_Contact(in1 := #Control_Screen_HMI, in2 := #Screen_5)
      Move(in := 12, out1 => #Control_Screen)
   END_RUNG
   RUNG wire#w4
      { S7_Templates := "SrcType := Word" } EQ_Contact(in1 := #Control_Screen_HMI, in2 := #Screen_6)
      Move(in := 13, out1 => #Control_Screen)
   END_RUNG
   RUNG wire#w4
      { S7_Templates := "SrcType := Word" } EQ_Contact(in1 := #Control_Screen_HMI, in2 := #Screen_8)
      Move(in := 14, out1 => #Control_Screen)
   END_RUNG
   // the same network as SCL:
   #_w1 := (((#Employee_Rework <> #Admin_1) AND (#Employee_Rework <> #Admin_2) AND (#Employee_Rework <> #Admin_3) AND (#Employee_Rework <> #Admin_4) AND (#Employee_Rework <> #Admin_5)) OR (#Employee_Rework = '')) AND (#Employee_Rework <> 'Lau') AND (#Control_Screen_HMI <> #Control_Screen);
   #_w2 := #_w1 AND #Everybody_Can_Access;
   IF #_w2 AND (#Control_Screen_HMI <> #Screen_10) THEN #Control_Screen := #Control_Screen_HMI; END_IF;
   IF #_w2 AND (#Control_Screen_HMI = #Screen_10) THEN #Control_Screen := 10; END_IF;
   #_w3 := #_w1 AND #Only_Admin_Can_Access;
   IF #_w3 AND (#Control_Screen_HMI = #Screen_4) THEN #Control_Screen := 11; END_IF;
   IF #_w3 AND (#Control_Screen_HMI = #Screen_5) THEN #Control_Screen := 12; END_IF;
   IF #_w3 AND (#Control_Screen_HMI = #Screen_6) THEN #Control_Screen := 13; END_IF;
   IF #_w3 AND (#Control_Screen_HMI = #Screen_8) THEN #Control_Screen := 14; END_IF;
END_REGION

REGION Network 4: Alarm
   RUNG wire#powerrail
      { S7_Templates := "SrcType := Word" } NE_Contact(in1 := #Alarm_0, in2 := 16#0)
      wire#w1
      P_Trig( #Aux_Trigger_10 )
      S_Coil( #Alarm )
   END_RUNG
   RUNG wire#powerrail
      { S7_Templates := "SrcType := Word" } NE_Contact(in1 := #Alarm_1, in2 := 16#0)
   END_RUNG wire#w1
   RUNG wire#powerrail
      { S7_Templates := "SrcType := Word" } NE_Contact(in1 := #Alarm_2, in2 := 16#0)
   END_RUNG wire#w1
   RUNG wire#powerrail
      { S7_Templates := "SrcType := Word" } EQ_Contact(in1 := #Alarm_0, in2 := 16#0)
      { S7_Templates := "SrcType := Word" } EQ_Contact(in1 := #Alarm_1, in2 := 16#0)
      { S7_Templates := "SrcType := Word" } EQ_Contact(in1 := #Alarm_2, in2 := 16#0)
      R_Coil( #Alarm )
   END_RUNG
   // the same network as SCL:
   #_w1 := (#Alarm_0 <> 16#0) OR (#Alarm_1 <> 16#0) OR (#Alarm_2 <> 16#0);
   #_w2 := #_w1 AND NOT #Aux_Trigger_10;   // rising edge
   #Aux_Trigger_10 := #_w1;
   IF #_w2 THEN #Alarm := TRUE; END_IF;
   IF (#Alarm_0 = 16#0) AND (#Alarm_1 = 16#0) AND (#Alarm_2 = 16#0) THEN #Alarm := FALSE; END_IF;
END_REGION

REGION Network 5
   RUNG wire#powerrail
      { S7_Templates := "SrcType := Word" } EQ_Contact(in1 := #Control_Screen, in2 := #Job_Mailbox[1])
      { S7_Templates := "SrcType := Word" } NE_Contact(in1 := #Job_Mailbox[0], in2 := 0)
      { S7_Templates := "time_type := Time" } #Timer_Delay_Change_Job_Mailbox.TON(pt := T#300MS, et =>)
      Move(in := 0, out1 => #Job_Mailbox[0])
   END_RUNG
   // the same network as SCL:
   #Timer_Delay_Change_Job_Mailbox(IN := (#Control_Screen = #Job_Mailbox[1]) AND (#Job_Mailbox[0] <> 0),   // TON
                           PT := T#300MS);
   IF #Timer_Delay_Change_Job_Mailbox.Q THEN #Job_Mailbox[0] := 0; END_IF;
END_REGION

REGION Network 6
   RUNG wire#powerrail
      { S7_Templates := "SrcType := Word" } NE_Contact(in1 := #Control_Screen, in2 := #Job_Mailbox[1])
      Move(in := 51, out1 => #Job_Mailbox[0])
      Move(in := 0, out1 => #Job_Mailbox[2], out2 => #Job_Mailbox[3])
      { S7_Templates := "time_type := Time" } #Timer_Delay_Change_Screen.TON(pt := T#200MS, et =>)
      Move(in := #Control_Screen, out1 => #Job_Mailbox[1])
   END_RUNG
   // the same network as SCL:
   #_w1 := #Control_Screen <> #Job_Mailbox[1];
   IF #_w1 THEN
       #Job_Mailbox[0] := 51;
       #Job_Mailbox[2] := 0;
       #Job_Mailbox[3] := 0;
   END_IF;
   #Timer_Delay_Change_Screen(IN := #_w1, PT := T#200MS);   // TON
   IF #Timer_Delay_Change_Screen.Q THEN #Job_Mailbox[1] := #Control_Screen; END_IF;
END_REGION
END_FUNCTION_BLOCK

FUNCTION_BLOCK "FB_IO_Device_Functional_Test_Rework"   // FB12, LAD
{ S7_Optimized_Access := 'TRUE' }
// stored: AutoNumber false, MemoryReserve 100, SetENOAutomatically false
   VAR_INPUT
      Reset_PLC_Functional_Test_Rework : Bool;
      Status : Bool;
      Voltage_Read : UInt;
      Min_Electrical_Current : UInt;
      Max_Electrical_Current : UInt;
      Time_End_Electrical_Current_Test : Time;
      Time_Start_Visual_Test : Time;
      In_Functional_Test_Rework : "IO_Device_Functinal_Test_Rework";
   END_VAR
   VAR_OUTPUT
      Out_Test_Parameters_Rework : "IO_Device_Test_Parameters_Rework";
      Comunication_Error_Panel_Rework : Bool;
   END_VAR
   VAR
      Timer_Alarme_A_1 { S7_SetPoint := 'True'} : TON_TIME;
      Timer_Alarme_B_1 { S7_SetPoint := 'True'} : TON_TIME;
   END_VAR
BEGIN

REGION Network 1
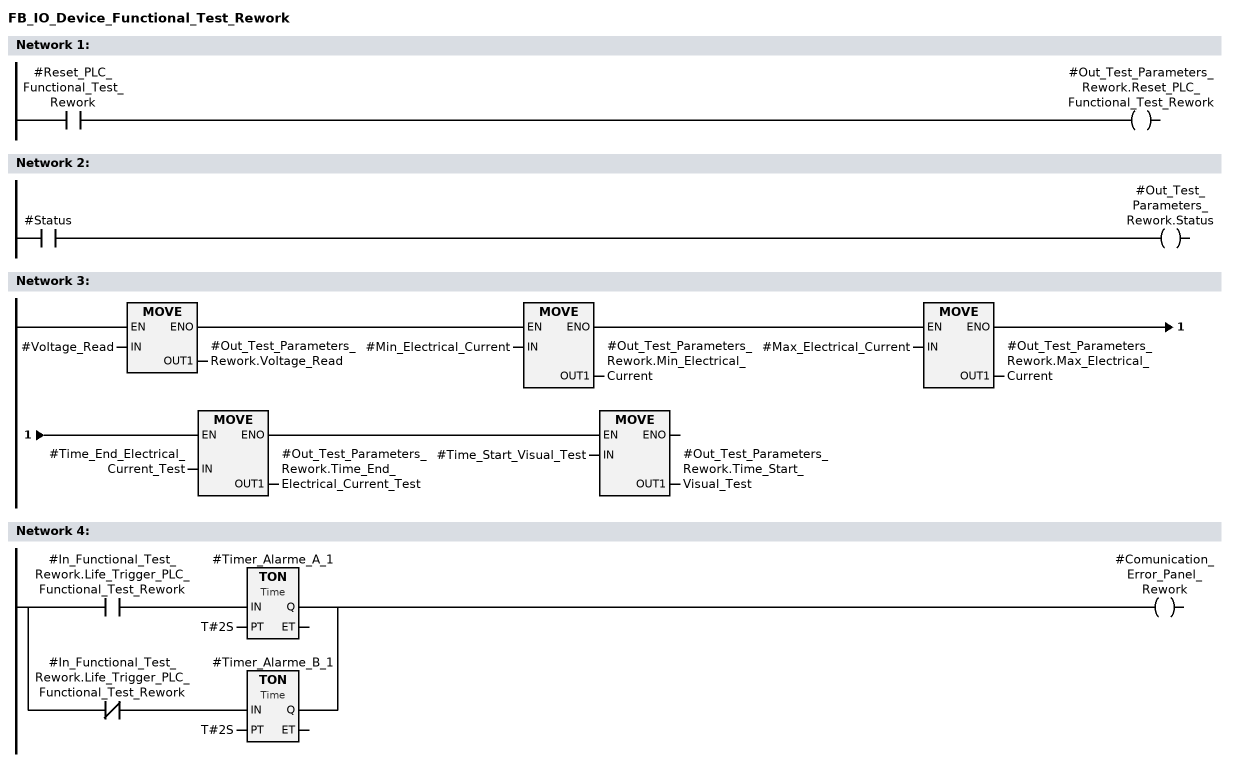
   RUNG wire#powerrail
      Contact( #Reset_PLC_Functional_Test_Rework )
      Coil( #Out_Test_Parameters_Rework.Reset_PLC_Functional_Test_Rework )
   END_RUNG
   // the same network as SCL:
   #Out_Test_Parameters_Rework.Reset_PLC_Functional_Test_Rework := #Reset_PLC_Functional_Test_Rework;
END_REGION

REGION Network 2
   RUNG wire#powerrail
      Contact( #Status )
      Coil( #Out_Test_Parameters_Rework.Status )
   END_RUNG
   // the same network as SCL:
   #Out_Test_Parameters_Rework.Status := #Status;
END_REGION

REGION Network 3
   RUNG wire#powerrail
      Move(in := #Voltage_Read, out1 => #Out_Test_Parameters_Rework.Voltage_Read)
      Move(in := #Min_Electrical_Current, out1 => #Out_Test_Parameters_Rework.Min_Electrical_Current)
      Move(in := #Max_Electrical_Current, out1 => #Out_Test_Parameters_Rework.Max_Electrical_Current)
      Move(in := #Time_End_Electrical_Current_Test, out1 => #Out_Test_Parameters_Rework.Time_End_Electrical_Current_Test)
      Move(in := #Time_Start_Visual_Test, out1 => #Out_Test_Parameters_Rework.Time_Start_Visual_Test)
   END_RUNG
   // the same network as SCL:
   #Out_Test_Parameters_Rework.Voltage_Read := #Voltage_Read;
   #Out_Test_Parameters_Rework.Min_Electrical_Current := #Min_Electrical_Current;
   #Out_Test_Parameters_Rework.Max_Electrical_Current := #Max_Electrical_Current;
   #Out_Test_Parameters_Rework.Time_End_Electrical_Current_Test := #Time_End_Electrical_Current_Test;
   #Out_Test_Parameters_Rework.Time_Start_Visual_Test := #Time_Start_Visual_Test;
END_REGION

REGION Network 4
   RUNG wire#powerrail
      Contact( #In_Functional_Test_Rework.Life_Trigger_PLC_Functional_Test_Rework )
      { S7_Templates := "time_type := Time" } #Timer_Alarme_A_1.TON(pt := T#2S, et =>)
      wire#w1
      Coil( #Comunication_Error_Panel_Rework )
   END_RUNG
   RUNG wire#powerrail
      I_Contact( #In_Functional_Test_Rework.Life_Trigger_PLC_Functional_Test_Rework )
      { S7_Templates := "time_type := Time" } #Timer_Alarme_B_1.TON(pt := T#2S, et =>)
   END_RUNG wire#w1
   // the same network as SCL:
   #Timer_Alarme_A_1(IN := #In_Functional_Test_Rework.Life_Trigger_PLC_Functional_Test_Rework, PT := T#2S);   // TON
   #Timer_Alarme_B_1(IN := NOT #In_Functional_Test_Rework.Life_Trigger_PLC_Functional_Test_Rework, PT := T#2S);   // TON
   #Comunication_Error_Panel_Rework := #Timer_Alarme_A_1.Q OR #Timer_Alarme_B_1.Q;
END_REGION
END_FUNCTION_BLOCK

ORGANIZATION_BLOCK "DiagnosticErrorInterrupt"   // OB82, LAD, DiagnosticErrorInterrupt
{ S7_Optimized_Access := 'TRUE' }
// stored: SetENOAutomatically false
   VAR_INPUT
      IO_State : Word;   // IO state of the HW object
      LADDR : HW_ANY;   // Hardware identifier
      Channel : UInt;   // Channel number
      MultiError : Bool;   // =true if more than one error is present
   END_VAR
BEGIN
END_ORGANIZATION_BLOCK

